stStationEvents[0].aEvents[25].bFault						:= TRUE;
stStationEvents[0].aEvents[25].bEventFlag					:= NOT stMachineStatus.bSystemPowerUp AND dw_T06_EL2904.stTerminalInfo.nTerminal_State <> 8;
stStationEvents[0].aEvents[25].bEventText					:= 'T06_EL2904 card in fault' ;
stStationEvents[0].aEvents[25].sSolution					:= 'Reset System';

stStationEvents[0].aEvents[26].bFault						:= TRUE;
stStationEvents[0].aEvents[26].bEventFlag					:= NOT stMachineStatus.bSystemPowerUp AND dw_T07_EL9410.stTerminalInfo.nTerminal_State <> 8;
stStationEvents[0].aEvents[26].bEventText					:= 'T07_EL9410 card in fault' ;
stStationEvents[0].aEvents[26].sSolution					:= 'Reset System';

stStationEvents[0].aEvents[27].bFault						:= TRUE;
stStationEvents[0].aEvents[27].bEventFlag					:= NOT stMachineStatus.bSystemPowerUp AND dw_T08_EL1809.stTerminalInfo.nTerminal_State <> 8;
stStationEvents[0].aEvents[27].bEventText					:= 'T08_EL1809 card in fault' ;
stStationEvents[0].aEvents[27].sSolution					:= 'Reset System';

stStationEvents[0].aEvents[28].bFault						:= TRUE;
stStationEvents[0].aEvents[28].bEventFlag					:= NOT stMachineStatus.bSystemPowerUp AND dw_T09_EL2809.stTerminalInfo.nTerminal_State <> 8;
stStationEvents[0].aEvents[28].bEventText					:= 'T09_EL2809 card in fault' ;
stStationEvents[0].aEvents[28].sSolution					:= 'Reset System';

stStationEvents[0].aEvents[29].bFault						:= TRUE;
stStationEvents[0].aEvents[29].bEventFlag					:= NOT stMachineStatus.bSystemPowerUp AND dw_T10_EL3058.stTerminalInfo.nTerminal_State <> 8;
stStationEvents[0].aEvents[29].bEventText					:= 'T10_EL3058 card in fault' ;
stStationEvents[0].aEvents[29].sSolution					:= 'Reset System';

stStationEvents[0].aEvents[30].bFault						:= TRUE;
stStationEvents[0].aEvents[30].bEventFlag					:= NOT stMachineStatus.bSystemPowerUp AND dw_T11_EL1918.stTerminalInfo.nTerminal_State <> 8;
stStationEvents[0].aEvents[30].bEventText					:= 'T11_EL1918 card in fault' ;
stStationEvents[0].aEvents[30].sSolution					:= 'Reset System';

stStationEvents[0].aEvents[31].bFault						:= TRUE;
stStationEvents[0].aEvents[31].bEventFlag					:= NOT stMachineStatus.bSystemPowerUp AND dw_T12_EL6633.stTerminalInfo.nTerminal_State <> 8 AND NOT abMachineDefinition[2];
stStationEvents[0].aEvents[31].bEventText					:= 'T12_EL6633 card in fault' ;
stStationEvents[0].aEvents[31].sSolution					:= 'Reset System';

//GENERAL
stStationEvents[0].aEvents[32].bFault						:= TRUE;
stStationEvents[0].aEvents[32].bEventFlag					:= bDoorClosingFlag AND (NOT dw_T05_EL1918.iLeftTouchButtonNO OR NOT dw_T05_EL1918.iRightTouchButtonNO);
stStationEvents[0].aEvents[32].bEventText					:= 'Hands out before door was closed' ;
stStationEvents[0].aEvents[32].sSolution					:= 'Reset System';

stStationEvents[0].aEvents[33].bFault						:= TRUE;
stStationEvents[0].aEvents[33].bEventFlag					:= ((stMachineStatus.eMachineState = E_MachineState.MANUAL_MODE) OR (stMachineStatus.eMachineState = E_MachineState.SYSTEM_AUTO_CYCLE ))
																AND bOutHMI;
stStationEvents[0].aEvents[33].bEventText					:= 'Out HMI while Machine was in Autocycle' ;
stStationEvents[0].aEvents[33].sSolution					:= 'Reset System';


stStationEvents[0].aEvents[34].bFault						:= TRUE;
stStationEvents[0].aEvents[34].bEventTimer(IN := (stMachineStatus.eMachineState = E_MachineState.SYSTEM_AUTO_CYCLE) AND NOT bAutocycleIDLE, PT := stTimers.tAutoCycleTimeOut );
stStationEvents[0].aEvents[34].bEventFlag					:= stStationEvents[0].aEvents[34].bEventTimer.Q;
stStationEvents[0].aEvents[34].bEventText					:= 'Auto Cycle Timeout' ;
stStationEvents[0].aEvents[34].sSolution					:= 'Reset System';

// PUCK LOCKER //Renan Added 06Jul26
stStationEvents[0].aEvents[35].bFault := stMACHINE.bPuckLocker;
stStationEvents[0].aEvents[35].bEventFlag := stMACHINE.bPuckLocker AND GVL_Stations.stPuckLocker.bUnexpectedRemovalFault;
stStationEvents[0].aEvents[35].bEventText := 'Puck removed while locker pin was engaged';
stStationEvents[0].aEvents[35].sSolution := 'Return puck to the locker position and acknowledge the alarm with Administrator access';





//STOP REQUEST

stStationEvents[0].aEvents[40].bCycleStopRequest			:= TRUE;
stStationEvents[0].aEvents[40].bEventFlag					:=  bOutHMI;
stStationEvents[0].aEvents[40].bEventText					:= 'Out HMI or User not logged in' ;
stStationEvents[0].aEvents[40].sSolution					:= '';

stStationEvents[0].aEvents[41].bCycleStopRequest			:= TRUE;
stStationEvents[0].aEvents[41].bEventTimer(IN := bAutocycleIDLE, PT := stTimers.tAutoCycleIDLETimeOut);
stStationEvents[0].aEvents[41].bEventFlag					:= stStationEvents[0].aEvents[41].bEventTimer.Q;
stStationEvents[0].aEvents[41].bEventText					:= 'Autocycle in IDLE Timeout' ;
stStationEvents[0].aEvents[41].sSolution					:= '';

stStationEvents[0].aEvents[42].bCycleStopRequest			:= TRUE;
stStationEvents[0].aEvents[42].bEventFlag					:= NOT dw_T08_EL1809.iStopButton;
stStationEvents[0].aEvents[42].bEventText					:= 'Stop Button Pressed' ;
stStationEvents[0].aEvents[42].sSolution					:= '';

stStationEvents[0].aEvents[43].bCycleStopRequest			:= TRUE;
stStationEvents[0].aEvents[43].bEventFlag					:=  stTwinSAFE.qMainDoorOpenned;
stStationEvents[0].aEvents[43].bEventText					:= 'Door openned ' ;
stStationEvents[0].aEvents[43].sSolution					:= 'Close door and Reset system to intilisation';


stStationEvents[0].aEvents[44].bCycleStopRequest			:= TRUE;
stStationEvents[0].aEvents[44].bEventFlag					:=  (stMachineStatus.eMachineState = E_MachineState.SYSTEM_AUTO_CYCLE) AND NOT bNest1Flag AND NOT bNest2Flag;
stStationEvents[0].aEvents[44].bEventText					:= 'No Nest enabled' ;
stStationEvents[0].aEvents[44].sSolution					:= 'Enable at least one Nest';


//MESSAGES

stStationEvents[0].aEvents[60].bMessage						:= TRUE;
stStationEvents[0].aEvents[60].bEventFlag					:=  bCSVError;
stStationEvents[0].aEvents[60].bEventText					:= 'CSV Not written ' ;
stStationEvents[0].aEvents[60].sSolution					:= '';
END_ACTION

END_PROGRAM

// ---- POUs/C_HMI/C_1_PRG_MainHMI.TcPOU
PROGRAM C_1_PRG_MainHMI
VAR
	
	bResetTest				: BOOL;
	i						: DINT;
	n						: DINT;//TABLE INDEX
	
	srRejectChuteFull			: SR; 

END_VAR

a_ACT_MachineStatusBaner();
b_ACT_Timers();
c_ACT_IO();

bEnableSettings				:= (stMachineStatus.eMachineState = E_MachineState.STOPPED);

stStatisticsWH[0]			:= stStatisticsHMI[0];
stStatisticsWH[1]			:= stStatisticsHMI[1];
stStatisticsWH[2]			:= stStatisticsHMI[4];
stStatisticsWH[3]			:= stStatisticsHMI[5];
stStatisticsWH[4]			:= stStatisticsHMI[6];
stStatisticsWH[5]			:= stStatisticsHMI[7];

stStatisticsLT[0]			:= stStatisticsHMI[0];
stStatisticsLT[1]			:= stStatisticsHMI[1];
stStatisticsLT[2]			:= stStatisticsHMI[2];
stStatisticsLT[3]			:= stStatisticsHMI[3];

bOpenRejectDialog			:= bRejectPartDialog[0] OR bRejectPartDialog[1] OR bRejectPartDialog[2];

bProcessCylinderDownEnable	:= dw_T08_EL1809.iPartPresentNest1 AND dw_T08_EL1809.iPartPresentNest2 AND dw_T05_EL1918.iProcessDoorFB;

srRejectChuteFull(SET1 := stStationEvents[0].aEvents[18].bEventTimer.Q, RESET := bEmptyRejectChuteAcknowledge AND NOT dw_T08_EL1809.iRejectSensor , Q1 => bEmptyRejectChute);

ACTION a_ACT_MachineStatusBaner:
//Machine status banner action
//SYSTEM POWER UP
IF stMachineStatus.bSystemPowerUp THEN	
	stStatusBanner.sMachineStatusText 							:= 'SYSTEM POWER UP';	
	stStatusBanner.nMachineStatusColour 						:= nWHITE;
	stStatusBanner.nMachineStatusTxtCol 						:= nBLACK;
	stStatusBanner.sBannerBckColor 								:= sWHITE;
	stStatusBanner.sBannerTextColor 							:= sBLACK;
END_IF

(* SYSTEM INITIALISING *)
IF stMachineStatus.bInitialising THEN	
	stStatusBanner.sMachineStatusText 							:= 'SYSTEM INITIALIZING';		
	stStatusBanner.nMachineStatusColour 						:= nYELLOW;
	stStatusBanner.nMachineStatusTxtCol 						:= nBLACK;
	stStatusBanner.sBannerBckColor 								:= sYELLOW;
	stStatusBanner.sBannerTextColor 							:= sBLACK;
END_IF

(* SAFETY *)
IF stMachineStatus.bSafety THEN	
	stStatusBanner.sMachineStatusText 							:= 'SYSTEM INITIALIZING';		
	stStatusBanner.nMachineStatusColour 						:= nYELLOW;
	stStatusBanner.nMachineStatusTxtCol 						:= nBLACK;
	stStatusBanner.sBannerBckColor 								:= sYELLOW;
	stStatusBanner.sBannerTextColor 							:= sBLACK;
END_IF


(* SYSTEM READY TO START FLASH ON *)
IF stMachineStatus.bReadyToStart AND stPuls.bFlash1Hz THEN
	stStatusBanner.sMachineStatusText 							:= 'SYSTEM READY TO START';		
	stStatusBanner.nMachineStatusColour 						:= nGREEN;
	stStatusBanner.nMachineStatusTxtCol 						:= nWHITE;
	stStatusBanner.sBannerBckColor 								:= sGREEN;
	stStatusBanner.sBannerTextColor 							:= sWHITE;
ELSIF stMachineStatus.bReadyToStart AND NOT stPuls.bFlash1Hz THEN	
	stStatusBanner.sMachineStatusText 							:= 'SYSTEM READY TO START';		
	stStatusBanner.nMachineStatusColour 						:= nWHITE;
	stStatusBanner.nMachineStatusTxtCol 						:= nGREEN;
	stStatusBanner.sBannerBckColor 								:= sWHITE;
	stStatusBanner.sBannerTextColor 							:= sGREEN;
END_IF

(* SYSTEM AUTO CYCLE *)
IF stMachineStatus.bAutoCycle THEN	
	stStatusBanner.sMachineStatusText 							:= 'SYSTEM AUTO CYCLE';		
	stStatusBanner.nMachineStatusColour 						:= nGREEN;
	stStatusBanner.nMachineStatusTxtCol 						:= nWHITE;
	stStatusBanner.sBannerBckColor 								:= sGREEN;
	stStatusBanner.sBannerTextColor 							:= sWHITE;	
END_IF

(* STOPPING *)
IF stMachineStatus.bStopping AND stPuls.bFlash1Hz THEN	
	stStatusBanner.sMachineStatusText 							:= 'STOPPING';		
	stStatusBanner.nMachineStatusColour 						:= nBLACK;
	stStatusBanner.nMachineStatusTxtCol 						:= nWHITE;
	stStatusBanner.sBannerBckColor 								:= sBLACK;
	stStatusBanner.sBannerTextColor 							:= sWHITE;	
ELSIF stMachineStatus.bStopping AND NOT stPuls.bFlash1Hz THEN	
	stStatusBanner.sMachineStatusText 							:= 'STOPPING';		
	stStatusBanner.nMachineStatusColour 						:= nWHITE;
	stStatusBanner.nMachineStatusTxtCol 						:= nBLACK;
	stStatusBanner.sBannerBckColor 								:= sWHITE;
	stStatusBanner.sBannerTextColor 							:= sBLACK;	
END_IF

(*STOPPED *)
IF stMachineStatus.bStopped THEN	
	stStatusBanner.sMachineStatusText 							:= 'CYCLE STOPPED';		
	stStatusBanner.nMachineStatusColour 						:= nBLACK;
	stStatusBanner.nMachineStatusTxtCol 						:= nWHITE;
	stStatusBanner.sBannerBckColor 								:= sBLACK;
	stStatusBanner.sBannerTextColor 							:= sWHITE;	
END_IF

(* FAULT FLASH ON *)
IF stMachineStatus.bFault AND stPuls.bFlash1Hz THEN	
	stStatusBanner.sMachineStatusText 							:= 'FAULT';		
	stStatusBanner.nMachineStatusColour 						:= nRED;
	stStatusBanner.nMachineStatusTxtCol 						:= nWHITE;
	stStatusBanner.sBannerBckColor 								:= sRED;
	stStatusBanner.sBannerTextColor 							:= sWHITE;	
ELSIF stMachineStatus.bFault AND NOT stPuls.bFlash1Hz THEN	
	stStatusBanner.sMachineStatusText 							:= 'FAULT';		
	stStatusBanner.nMachineStatusColour 						:= nWHITE;
	stStatusBanner.nMachineStatusTxtCol 						:= nBLACK;
	stStatusBanner.sBannerBckColor 								:= sWHITE;
	stStatusBanner.sBannerTextColor 							:= sBLACK;	
END_IF

(* MANUAL MODE *)
IF stMachineStatus.bManualMode THEN	
	stStatusBanner.sMachineStatusText 							:= 'MANUAL MODE';		
	stStatusBanner.nMachineStatusColour 						:= nBLUE;
	stStatusBanner.nMachineStatusTxtCol 						:= nWHITE;
	stStatusBanner.sBannerBckColor 								:= sBLUE;
	stStatusBanner.sBannerTextColor 							:= sWHITE;	
END_IF
END_ACTION

ACTION b_ACT_Timers:

stTimers.tAutoCycleTimeOut		:= DINT_TO_TIME(stTimers.nAutoCycleTimeOut * 1000) ;
stTimers.tDoorOpenedSignal		:= DINT_TO_TIME(stTimers.nDoorOpenedSignal * 1000) ;
stTimers.tStation1TimeOut		:= DINT_TO_TIME(stTimers.nStation1TimeOut * 1000) ;
stTimers.tStation2TimeOut		:= DINT_TO_TIME(stTimers.nStation2TimeOut * 1000) ;
stTimers.tStation3TimeOut		:= DINT_TO_TIME(stTimers.nStation3TimeOut * 1000) ;
stTimers.tTwoHandsSignal		:= DINT_TO_TIME(stTimers.nTwoHandsSignal * 1000) ;
stTimers.tHeightTest			:= DINT_TO_TIME(stTimers.nHeightTest * 1000) ;
stTimers.tAutoCycleIDLETimeOut			:= DINT_TO_TIME(stTimers.nAutoCycleIDLETimeOut * 1000) ;
END_ACTION

ACTION c_ACT_IO:
dw_T09_EL2809.qPanelLightLED				:= bLightsOnOff;
END_ACTION

END_PROGRAM

// ---- POUs/Utilities/PRG_Puls.TcPOU
PROGRAM PRG_Puls
VAR
	    //=== Master Pulses ===//
	fbScalingFlash  :FB_Pulse;
	fbScalingFlash4 :FB_Pulse;
	fbScalingFlash5 :FB_Pulse;
	fbFlash100Hz    :FB_Pulse;
	fbFlash10Hz		:FB_Pulse;
	fbFlash10HzB    :FB_Pulse;
	fbFlash4Hz		:FB_Pulse;
	fbFlash2Hz		:FB_Pulse;
	fbFlash1Hz		:FB_Pulse;
    fbFlash5Sec     :FB_Pulse;			

END_VAR

    //=== Master Pulses ===//
(**************************************************************************************************)
fbScalingFlash(
	bEnable	:=	TRUE,
	tPulseOn	:=	T#2MS,
	tPulseOff	:=	T#2MS,
	bFlash		=>	stPuls.bFlashScale
);

fbScalingFlash4(
     bEnable	:=	TRUE,
	tPulseOn	:=	T#4MS,
	tPulseOff	:=	T#4MS,
	bFlash		=>	stPuls.bFlashScale4
);
fbScalingFlash5(
     bEnable	:=	TRUE,
	tPulseOn	:=	T#5MS,
	tPulseOff	:=	T#5MS,
	bFlash		=>	stPuls.bFlashScale5
);



fbFlash100Hz(
	bEnable	:=	TRUE,
	tPulseOn	:=	T#10MS,
	tPulseOff	:=	T#10MS,
	bFlash		=>	stPuls.bFlash100Hz
);


fbFlash10HzB ( 
    bEnable	    :=	TRUE,
	tPulseOn	:=	T#20MS,//  T#50MS,
	tPulseOff	:=	T#20MS,//  T#50MS,
	bFlash		=>	stPuls.bFlash10BHz
);


fbFlash10Hz(
	bEnable	:=	TRUE,
	tPulseOn	:=	T#100MS,
	tPulseOff	:=	T#100MS,
	bFlash		=>	stPuls.bFlash10Hz
);


fbFlash4Hz(
	bEnable	:=	TRUE,
	tPulseOn	:=	T#250MS,
	tPulseOff	:=	T#250MS,
	bFlash		=>	stPuls.bFlash4Hz
);

fbFlash2Hz(
	bEnable	:=	TRUE,
	tPulseOn	:=	T#500MS,
	tPulseOff	:=	T#500MS,
	bFlash		=>	stPuls.bFlash2Hz
);

fbFlash1Hz(
	bEnable	:=	TRUE,
	tPulseOn	:=	T#1000MS,
	tPulseOff	:=	T#1000MS,
	bFlash		=>	stPuls.bFlash1Hz
);

fbFlash5Sec(
	bEnable	:=	TRUE,
	tPulseOn	:=	T#5S,
	tPulseOff	:=	T#5S,
	bFlash		=>	stPuls.bFlash5sec
);

END_PROGRAM

// ---- POUs/Utilities/FB_Pulse.TcPOU
FUNCTION_BLOCK FB_Pulse
VAR_INPUT
	bEnable		    :	BOOL;
	tPulseOn		:	TIME;
	tPulseOff		:	TIME;
END_VAR
VAR_OUTPUT
	bFlash			:	BOOL;
END_VAR
VAR
	tonFlashOn		:	TON;
	tonFlashOff	    :	TON;
END_VAR

IF 		(bEnable 	AND NOT 	tonFlashOff.Q)		THEN
	tonFlashOn.IN			:=	TRUE;
ELSE
	tonFlashOn.IN			:=	FALSE;
END_IF

tonFlashOn(
	IN:= ,
	PT:= tPulseOn,
	Q=> ,
	ET=>
);
tonFlashOff(
	IN:= tonFlashOn.Q,
	PT:= tPulseOff,
	Q=> ,
	ET=>
);

bFlash	:=	tonFlashOn.Q;

END_FUNCTION_BLOCK

// ---- POUs/B_STATIONS/B_2_HEIGHT_TEST/B_2_1_PRG_Master_Height_Test.TcPOU
PROGRAM B_2_1_PRG_Master_Height_Test

VAR

	rGoodStatistics						: ARRAY[0..1] OF  R_TRIG;
	rBadStatistics						: ARRAY[0..1] OF  R_TRIG;
	rEfficency							: STRING(510);
	
	anMinimumDistance					: ARRAY[1..3] OF REAL;
	anMaximumDistance					: ARRAY[1..3] OF REAL;

/////////////////////////////////////////////////////////////////////////////////////I O/////////////////////////////////////////////////////////////////////////////////////	
	
	abPass1								: ARRAY [1..3] OF BOOL;
	abFail1								: ARRAY [1..3] OF BOOL;
	abPass2								: ARRAY [1..3] OF BOOL;
	abFail2								: ARRAY [1..3] OF BOOL;
	tonTakeMeasure						: TON;
	abMeaurement						: ARRAY [0..1] OF BOOL;
	bMeasurementDone					: BOOL;

	abProbeError1						: ARRAY[1..4] OF BOOL;
	abProbeError2						: ARRAY[1..4] OF BOOL;
	bGeneralProbeError					: BOOL;
	bGeneralError						: BOOL;
	anRawMesurement1					: ARRAY[1..4] OF REAL;
	anRawMesurement2					: ARRAY[1..4] OF REAL;
	anRealDistance1						: ARRAY[1..3] OF REAL;
	anRealDistance2						: ARRAY[1..3] OF REAL;
	(*Renan - Added on 30Jun2026 *)
	anCorrectedMeasurement1 			: ARRAY [1..4] OF REAL;
    anCorrectedMeasurement2 			: ARRAY [1..4] OF REAL;
	(*/Renan - Added on 30Jun2026 *)

	i									: DINT;
	j									: DINT; //Index for settings
	
	
	

	
END_VAR

d_ACT_Set_Events_Station_2();
a_ACT_Ctrl_Station_2();
b_ACT_IO();
c_ACT_Statistics_Station_2();
e_ACT_Measurement();
f_ACT_ManualMode();
g_ACT_Settings();

ACTION a_ACT_Ctrl_Station_2:
/////////////////////////////////////////////////////////////////////////////////////UTILITIES/////////////////////////////////////////////////////////////////////////////////////
IF bGeneralProbeError OR bGeneralError OR stHeightTests.CMD.bAbort THEN
	
	stHeightTests.State			:= E_HeightTest_State.RESET;

ELSIF stHeightTests.CMD.bManualMode THEN
	
	stHeightTests.State			:= E_HeightTest_State.MANUAL_MODE;
	
END_IF



/////////////////////////////////////////////////////////////////////////////////////CONDITIONS/////////////////////////////////////////////////////////////////////////////////////

CASE stHeightTests.State OF
	
	E_HeightTest_State.ABORTED:

								IF 	stHeightTests.CMD.bEnable THEN
									
									stHeightTests.State			:= E_HeightTest_State.READY;
								
								END_IF
								
								

	E_HeightTest_State.READY:
	
								IF stHeightTests.CMD.bExecute THEN
									
									stHeightTests.State			:= E_HeightTest_State.MEASURE;
								
								END_IF
		
	E_HeightTest_State.MEASURE:				
									
								IF stHeightTests.CMD.HeightTest_CMD.Measurement1 AND stHeightTests.CMD.HeightTest_CMD.Measurement2 THEN
										
									abMeaurement[0]			:= TRUE;
									abMeaurement[1]			:= TRUE;
									
								ELSIF stHeightTests.CMD.HeightTest_CMD.Measurement1 AND NOT stHeightTests.CMD.HeightTest_CMD.Measurement2 THEN
									
									abMeaurement[0]			:= TRUE;
									
								ELSIF NOT stHeightTests.CMD.HeightTest_CMD.Measurement1 AND stHeightTests.CMD.HeightTest_CMD.Measurement2 THEN
									
									abMeaurement[1]			:= TRUE;
									
								END_IF
									
								stHeightTests.State			:= E_HeightTest_State.WAIT_MEASUREMENT;
								
	E_HeightTest_State.WAIT_MEASUREMENT:						
								
								e_ACT_Measurement();
								
								IF stHeightTests.CMD.HeightTest_CMD.Measurement1 THEN
									
									stCycleDataNest1.HeightTest_anRawMeasurement				:= anRawMesurement1;
									stCycleDataNest1.HeightTest_anDistancesResult 				:= anRealDistance1;
									stCycleDataNest1.HeightTest_bDistancesResult				:= abPass1;
									
								END_IF
								IF stHeightTests.CMD.HeightTest_CMD.Measurement2 THEN
									
									stCycleDataNest2.HeightTest_anRawMeasurement				:= anRawMesurement2;																
									stCycleDataNest2.HeightTest_anDistancesResult 				:= anRealDistance2;																
									stCycleDataNest2.HeightTest_bDistancesResult				:= abPass2;
									
								END_IF
								
								
								IF bMeasurementDone THEN
			
									stHeightTests.State		:= E_HeightTest_State.DONE;
								
								END_IF
										
	E_HeightTest_State.DONE:
								IF  stHeightTests.CMD.bAcknowledge THEN
									
									stHeightTests.State									:= E_HeightTest_State.RESULTS;
									stHeightTests.CMD.bAcknowledge 						:= FALSE;
									
								END_IF	
								
	E_HeightTest_State.RESULTS:
							
								IF abMeaurement[0] THEN
									IF abPass1[1] AND abPass1[2] AND abPass1[3] THEN
									
										stCycleDataNest1.HeightTest_Pass				:= TRUE;
									
									ELSE stCycleDataNest1.HeightTest_Fail 				:= TRUE;
								
									END_IF
								END_IF
								
								IF abMeaurement[1] THEN
									IF abPass2[1] AND abPass2[2] AND abPass2[3] THEN
									
										stCycleDataNest2.HeightTest_Pass				:= TRUE;
									
									ELSE stCycleDataNest2.HeightTest_Fail  			:= TRUE;
								
									END_IF
								END_IF	
								
								stHeightTests.State										:= E_HeightTest_State.RESET;
								
	E_HeightTest_State.RESET:
	
								abMeaurement[0]											:= FALSE;
								abMeaurement[1]											:= FALSE;
								bMeasurementDone										:= FALSE;

								FOR i := 1 TO 3 DO
									
									abPass1[i]											:= FALSE;
									abFail1[i]											:= FALSE;
									abPass2[i]											:= FALSE;
									abFail2[i]											:= FALSE;
								
								END_FOR
								
								IF bGeneralProbeError OR bGeneralError THEN
									
									stHeightTests.State									:= E_HeightTest_State.ERROR;
								
								ELSIF stHeightTests.CMD.bAbort THEN
									
									stHeightTests.State									:= E_HeightTest_State.ABORTED;
								
								ELSE stHeightTests.State								:= E_HeightTest_State.READY;
									
								END_IF
								
								
	
	E_HeightTest_State.ERROR:
	
								IF NOT bGeneralProbeError OR bGeneralError THEN
									
									stHeightTests.State									:= E_HeightTest_State.RESET;
									
								END_IF
							
	E_HeightTest_State.MANUAL_MODE:
	
								f_ACT_ManualMode();
								
								IF NOT stHeightTests.CMD.bManualMode THEN
									
									stHeightTests.State									:= E_HeightTest_State.ABORTED;
									
								END_IF
								
	
								

ELSE stHeightTests.State := E_HeightTest_State.READY;
	
END_CASE
/////////////////////////////////////////////////////////////////////////////////////STATUS/////////////////////////////////////////////////////////////////////////////////////

stHeightTests.Status.bBusy	:= 	stHeightTests.State	= E_HeightTest_State.WAIT_MEASUREMENT;	

stHeightTests.Status.bDone	:= 	stHeightTests.State	= E_HeightTest_State.DONE;

stHeightTests.Status.bError	:= 	stHeightTests.State	= E_HeightTest_State.ERROR;	

stHeightTests.Status.bReady	:=	stHeightTests.State	= E_HeightTest_State.READY;

stHeightTests.Status.bStopped := NOT stHeightTests.Status.bBusy;
END_ACTION

ACTION b_ACT_IO:

	abProbeError1					:= Probes.stProbesSet[1].abProbeError;
	abProbeError2					:= Probes.stProbesSet[2].abProbeError;
	bGeneralError					:= Probes.bGeneralError;
	anRawMesurement1				:= Probes.stProbesSet[1].anScaledRawMeasurement;
	anRawMesurement2				:= Probes.stProbesSet[2].anScaledRawMeasurement;
	


	bGeneralProbeError				:= 	abProbeError1[1] OR abProbeError1[2] OR abProbeError1[3] OR abProbeError1[4] OR
										abProbeError2[1] OR abProbeError2[2] OR abProbeError2[3] OR abProbeError2[4];
										
	stCycleDataNest1.HeightTest_anSetPoint := stProbesSettings.anExpectedDistances;
	stCycleDataNest2.HeightTest_anSetPoint := stProbesSettings.anExpectedDistances;
END_ACTION

ACTION c_ACT_Statistics_Station_2:
stStatisticsHMI[4].sName			:= 'Height Test 1';
stStatisticsHMI[5].sName			:= 'Height Test 2';


rGoodStatistics[0]( CLK := stCycleDataNest1.HeightTest_Pass);
rGoodStatistics[1]( CLK := stCycleDataNest2.HeightTest_Pass);
rBadStatistics[0]	( CLK := stCycleDataNest1.HeightTest_Fail);
rBadStatistics[1]	( CLK := stCycleDataNest2.HeightTest_Fail);

//statistics 1
IF 	rGoodStatistics[0].Q THEN
	
	stStatisticsHMI[4].nGood		:= stStatisticsHMI[4].nGood + 1;
	
END_IF
								
IF 	rBadStatistics[0].Q THEN
	
	stStatisticsHMI[4].nBad			:= stStatisticsHMI[4].nBad + 1;
	
END_IF

IF stStatisticsHMI[4].bResetGood THEN
	stStatisticsHMI[4].nGood		:= 0;
END_IF

IF stStatisticsHMI[4].bResetBad THEN
	stStatisticsHMI[4].nBad			:= 0;
END_IF

IF (( stStatisticsHMI[4].nGood + stStatisticsHMI[4].nBad) <> 0) THEN
	
	rEfficency							:= LREAL_TO_FMTSTR(in := (DINT_TO_REAL(stStatisticsHMI[4].nGood) /( DINT_TO_REAL(stStatisticsHMI[4].nGood) + DINT_TO_REAL(stStatisticsHMI[4].nBad))) * 100.0,iPrecision := 2, bRound := TRUE);
	stStatisticsHMI[4].nEfficency		:= CONCAT(STR1 := '%', STR2 := (rEfficency));

ELSE stStatisticsHMI[4].nEfficency		:= CONCAT(STR1 := '%', STR2 := (DINT_TO_STRING(0)));
	
END_IF
//statistics 2
IF 	rGoodStatistics[1].Q THEN
	
	stStatisticsHMI[5].nGood		:= stStatisticsHMI[5].nGood + 1;
	
END_IF
								
IF 	rBadStatistics[1].Q THEN
	
	stStatisticsHMI[5].nBad			:= stStatisticsHMI[5].nBad + 1;
	
END_IF

IF stStatisticsHMI[5].bResetGood THEN
	stStatisticsHMI[5].nGood		:= 0;
END_IF

IF stStatisticsHMI[5].bResetBad THEN
	stStatisticsHMI[5].nBad			:= 0;
END_IF

IF (( stStatisticsHMI[5].nGood + stStatisticsHMI[5].nBad) <> 0) THEN
	
	rEfficency							:= LREAL_TO_FMTSTR(in := (DINT_TO_REAL(stStatisticsHMI[5].nGood) /( DINT_TO_REAL(stStatisticsHMI[5].nGood) + DINT_TO_REAL(stStatisticsHMI[5].nBad))) * 100.0,iPrecision := 2, bRound := TRUE);
	stStatisticsHMI[5].nEfficency		:= CONCAT(STR1 := '%', STR2 := (rEfficency));

ELSE stStatisticsHMI[5].nEfficency		:= CONCAT(STR1 := '%', STR2 := (DINT_TO_STRING(0)));
	
END_IF
END_ACTION

ACTION d_ACT_Set_Events_Station_2:
//FAULTS

stStationEvents[2].aEvents[0].bFault						:= TRUE;
stStationEvents[2].aEvents[0].bEventFlag					:= bGeneralError;
stStationEvents[2].aEvents[0].bEventText					:= 'Probes general error';
stStationEvents[2].aEvents[0].sSolution						:= 'Check probes amplifier and ethercat unit';

stStationEvents[2].aEvents[1].bFault						:= TRUE;
stStationEvents[2].aEvents[1].bEventFlag					:= abProbeError1[1];
stStationEvents[2].aEvents[1].bEventText					:= 'Probes 1 error';
stStationEvents[2].aEvents[1].sSolution						:= 'Check probe 1';

stStationEvents[2].aEvents[2].bFault						:= TRUE;
stStationEvents[2].aEvents[2].bEventFlag					:= abProbeError1[2];
stStationEvents[2].aEvents[2].bEventText					:= 'Probes 2 error';
stStationEvents[2].aEvents[2].sSolution						:= 'Check probe 2';

stStationEvents[2].aEvents[3].bFault						:= TRUE;
stStationEvents[2].aEvents[3].bEventFlag					:= abProbeError1[3];
stStationEvents[2].aEvents[3].bEventText					:= 'Probes 3 error';
stStationEvents[2].aEvents[3].sSolution						:= 'Check probe 3';

stStationEvents[2].aEvents[4].bFault						:= TRUE;
stStationEvents[2].aEvents[4].bEventFlag					:= abProbeError1[4];
stStationEvents[2].aEvents[4].bEventText					:= 'Probes 4 error';
stStationEvents[2].aEvents[4].sSolution						:= 'Check probe 4';

stStationEvents[2].aEvents[5].bFault						:= TRUE;
stStationEvents[2].aEvents[5].bEventFlag					:= abProbeError2[1];
stStationEvents[2].aEvents[5].bEventText					:= 'Probes 5 error';
stStationEvents[2].aEvents[5].sSolution						:= 'Check probe 5';

stStationEvents[2].aEvents[6].bFault						:= TRUE;
stStationEvents[2].aEvents[6].bEventFlag					:= abProbeError2[2];
stStationEvents[2].aEvents[6].bEventText					:= 'Probes 6 error';
stStationEvents[2].aEvents[6].sSolution						:= 'Check probe 6';

stStationEvents[2].aEvents[7].bFault						:= TRUE;
stStationEvents[2].aEvents[7].bEventFlag					:= abProbeError2[3];
stStationEvents[2].aEvents[7].bEventText					:= 'Probes 7 error';
stStationEvents[2].aEvents[7].sSolution						:= 'Check probe 7';

stStationEvents[2].aEvents[8].bFault						:= TRUE;
stStationEvents[2].aEvents[8].bEventFlag					:= abProbeError2[4];
stStationEvents[2].aEvents[8].bEventText					:= 'Probes 8 error';
stStationEvents[2].aEvents[8].sSolution						:= 'Check probe 8';

stStationEvents[2].aEvents[9].bFault						:= TRUE;
stStationEvents[2].aEvents[9].bEventTimer(IN := stHeightTests.Status.bBusy, PT := stTimers.tStation2TimeOut);
stStationEvents[2].aEvents[9].bEventFlag					:= stStationEvents[2].aEvents[9].bEventTimer.Q;
stStationEvents[2].aEvents[9].bEventText					:= 'Height test cycle Timeout';
stStationEvents[2].aEvents[9].sSolution						:= 'Reset System';
END_ACTION

ACTION e_ACT_Measurement:

tonTakeMeasure(IN:= stHeightTests.State = E_HeightTest_State.WAIT_MEASUREMENT, PT := stTimers.tHeightTest);

IF tonTakeMeasure.Q THEN
	
	IF abMeaurement[0] THEN
	
		FOR i := 1 TO 3 DO
		
			IF (anRealDistance1[i] > anMinimumDistance[i]) AND (anRealDistance1[i] < anMaximumDistance[i]) THEN
		
				abPass1[i]						:= TRUE;
			
			ELSE abFail1[i]						:= TRUE;	
				
			END_IF
		
		END_FOR

	END_IF
	
	IF abMeaurement[1] THEN
	
		FOR i := 1 TO 3 DO
		
			IF (anRealDistance2[i] > anMinimumDistance[i]) AND (anRealDistance2[i] < anMaximumDistance[i]) THEN
		
				abPass2[i]						:= TRUE;
			
			ELSE abFail2[i]						:= TRUE;	
				
			END_IF
		
		END_FOR

	END_IF

	bMeasurementDone							:= TRUE;
	i											:= 0;
END_IF
END_ACTION

ACTION f_ACT_ManualMode:
IF stPuls.bFlash100Hz THEN
	
	FOR i := 1 TO 3 DO
		
		IF (anRealDistance1[i] > anMinimumDistance[i]) AND (anRealDistance1[i] < anMaximumDistance[i]) THEN
		
			stAnimations.abDistanceBoxesGreen[i]	:= TRUE;
			
		ELSE stAnimations.abDistanceBoxesGreen[i]	:= FALSE;	
				
		END_IF
		
	END_FOR
	i												:= 0;
	FOR i := 1 TO 3 DO
		
		IF (anRealDistance2[i] > anMinimumDistance[i]) AND (anRealDistance2[i] < anMaximumDistance[i]) THEN
		
			stAnimations.abDistanceBoxesGreen[3+i]	:= TRUE;
			
		ELSE stAnimations.abDistanceBoxesGreen[3+i]	:= FALSE;	
				
		END_IF
		
	END_FOR
	
	i												:= 0;
END_IF
END_ACTION

ACTION g_ACT_Settings:
//settings tolerances

anMinimumDistance[1]					:= stProbesSettings.anExpectedDistances[1] - stProbesSettings.anTolerances[1];//settings from HMI
anMaximumDistance[1]					:= stProbesSettings.anExpectedDistances[1] + stProbesSettings.anTolerances[1];//settings from HMI
anMinimumDistance[2]					:= stProbesSettings.anExpectedDistances[2] - stProbesSettings.anTolerances[2];//settings from HMI
anMaximumDistance[2]					:= stProbesSettings.anExpectedDistances[2] + stProbesSettings.anTolerances[2];//settings from HMI
anMinimumDistance[3]					:= stProbesSettings.anExpectedDistances[3] - stProbesSettings.anTolerances[3];//settings from HMI
anMaximumDistance[3]					:= stProbesSettings.anExpectedDistances[3] + stProbesSettings.anTolerances[3];//settings from HMI





//setting the bit according to the probe from bit 1 to bit 8
IF abPresetProbe[1] THEN
	
	Probes.abPresetProbe						:= 2;

ELSIF abPresetProbe[2] THEN
	
	Probes.abPresetProbe						:= 4;
	
ELSIF abPresetProbe[3] THEN
	
	Probes.abPresetProbe						:= 8;
	
ELSIF abPresetProbe[4] THEN
	
	Probes.abPresetProbe						:= 16;
	
ELSIF abPresetProbe[5] THEN
	
	Probes.abPresetProbe						:= 32;
	
ELSIF abPresetProbe[6] THEN
	
	Probes.abPresetProbe						:= 64;
	
ELSIF abPresetProbe[7] THEN
	
	Probes.abPresetProbe						:= 128;
	
ELSIF abPresetProbe[8] THEN
	
	Probes.abPresetProbe						:= 256;

END_IF

Probes.stProbesSet[1].anScaledRawMeasurement[1]					:= DINT_TO_REAL(Probes.stProbesSet[1].anRawMeasurement[1])/10000;
Probes.stProbesSet[1].anScaledRawMeasurement[2]					:= DINT_TO_REAL(Probes.stProbesSet[1].anRawMeasurement[2])/10000;
Probes.stProbesSet[1].anScaledRawMeasurement[3]					:= DINT_TO_REAL(Probes.stProbesSet[1].anRawMeasurement[3])/10000;
Probes.stProbesSet[1].anScaledRawMeasurement[4]					:= DINT_TO_REAL(Probes.stProbesSet[1].anRawMeasurement[4])/10000;

Probes.stProbesSet[2].anScaledRawMeasurement[1]					:= DINT_TO_REAL(Probes.stProbesSet[2].anRawMeasurement[1])/10000;
Probes.stProbesSet[2].anScaledRawMeasurement[2]					:= DINT_TO_REAL(Probes.stProbesSet[2].anRawMeasurement[2])/10000;
Probes.stProbesSet[2].anScaledRawMeasurement[3]					:= DINT_TO_REAL(Probes.stProbesSet[2].anRawMeasurement[3])/10000;
Probes.stProbesSet[2].anScaledRawMeasurement[4]					:= DINT_TO_REAL(Probes.stProbesSet[2].anRawMeasurement[4])/10000;

IF Probes.stProbesSet[1].anScaledRawMeasurement[1] > 2 AND Probes.stProbesSet[1].anScaledRawMeasurement[1] < 12 AND 
	Probes.stProbesSet[1].anScaledRawMeasurement[2] > 2 AND Probes.stProbesSet[1].anScaledRawMeasurement[2] < 12 AND 
	Probes.stProbesSet[1].anScaledRawMeasurement[3] > 2 AND Probes.stProbesSet[1].anScaledRawMeasurement[3] < 12 AND 
	Probes.stProbesSet[1].anScaledRawMeasurement[4] > 2 AND Probes.stProbesSet[1].anScaledRawMeasurement[4] < 12 THEN 
	
	bEnableSetCablibrationBlock1								:= TRUE;
	
ELSE bEnableSetCablibrationBlock1								:= FALSE;
	
END_IF

IF Probes.stProbesSet[2].anScaledRawMeasurement[1] > 2 AND Probes.stProbesSet[2].anScaledRawMeasurement[1] < 12 AND 
	Probes.stProbesSet[2].anScaledRawMeasurement[2] > 2 AND Probes.stProbesSet[2].anScaledRawMeasurement[2] < 12 AND 
	Probes.stProbesSet[2].anScaledRawMeasurement[3] > 2 AND Probes.stProbesSet[2].anScaledRawMeasurement[3] < 12 AND 
	Probes.stProbesSet[2].anScaledRawMeasurement[4] > 2 AND Probes.stProbesSet[2].anScaledRawMeasurement[4] < 12 THEN 
	
	bEnableSetCablibrationBlock2								:= TRUE;
	
ELSE bEnableSetCablibrationBlock2								:= FALSE;
	
END_IF

//calibration block
IF bSetCalibrationBlock1 THEN
	
	stProbesSettings.anHeightSetByCalibration1[1]				:= Probes.stProbesSet[1].anScaledRawMeasurement[1];
	stProbesSettings.anHeightSetByCalibration1[2]				:= Probes.stProbesSet[1].anScaledRawMeasurement[2];
	stProbesSettings.anHeightSetByCalibration1[3]				:= Probes.stProbesSet[1].anScaledRawMeasurement[3];
	stProbesSettings.anHeightSetByCalibration1[4]				:= Probes.stProbesSet[1].anScaledRawMeasurement[4];
	
	stProbesSettings.nDistanceOffset1[1]						:= stProbesSettings.anDistanceCalibrationBlock[1] - (Probes.stProbesSet[1].anScaledRawMeasurement[2] - Probes.stProbesSet[1].anScaledRawMeasurement[1]);
	stProbesSettings.nDistanceOffset1[2]						:= stProbesSettings.anDistanceCalibrationBlock[2] - (Probes.stProbesSet[1].anScaledRawMeasurement[3] - Probes.stProbesSet[1].anScaledRawMeasurement[1]);
	stProbesSettings.nDistanceOffset1[3]						:= stProbesSettings.anDistanceCalibrationBlock[3] - (Probes.stProbesSet[1].anScaledRawMeasurement[4] - Probes.stProbesSet[1].anScaledRawMeasurement[1]);
	
END_IF



IF bSetCalibrationBlock2 THEN
	
	stProbesSettings.anHeightSetByCalibration2[1]				:= Probes.stProbesSet[2].anScaledRawMeasurement[1];
	stProbesSettings.anHeightSetByCalibration2[2]				:= Probes.stProbesSet[2].anScaledRawMeasurement[2];
	stProbesSettings.anHeightSetByCalibration2[3]				:= Probes.stProbesSet[2].anScaledRawMeasurement[3];
	stProbesSettings.anHeightSetByCalibration2[4]				:= Probes.stProbesSet[2].anScaledRawMeasurement[4];
	
	stProbesSettings.nDistanceOffset2[1]						:= stProbesSettings.anDistanceCalibrationBlock[1] - (Probes.stProbesSet[2].anScaledRawMeasurement[2] - Probes.stProbesSet[2].anScaledRawMeasurement[1]);
	stProbesSettings.nDistanceOffset2[2]						:= stProbesSettings.anDistanceCalibrationBlock[2] - (Probes.stProbesSet[2].anScaledRawMeasurement[3] - Probes.stProbesSet[2].anScaledRawMeasurement[1]);
	stProbesSettings.nDistanceOffset2[3]						:= stProbesSettings.anDistanceCalibrationBlock[3] - (Probes.stProbesSet[2].anScaledRawMeasurement[4] - Probes.stProbesSet[2].anScaledRawMeasurement[1]);

END_IF

(* Renan Added 30Jun26 - Nest offset by probe *)
IF bSetProbeOffsetNest1 THEN
	FOR i := 1 TO 4 DO
		stProbesSettings.anNestOffsetByProbe1[i] := anNestOffsetByProbe1[i];
		stProbesSettings.anNestOffsetByProbe2[i] := anNestOffsetByProbe2[i];
	END_FOR
	bSetProbeOffsetNest1 := FALSE;
END_IF

FOR i := 1 TO 4 DO
    anCorrectedMeasurement1[i] := Probes.stProbesSet[1].anScaledRawMeasurement[i] + stProbesSettings.anNestOffsetByProbe1[i];
    anCorrectedMeasurement2[i] := Probes.stProbesSet[2].anScaledRawMeasurement[i] + stProbesSettings.anNestOffsetByProbe2[i];
END_FOR

(* Renan Changed 30Jun26 - Nest offset by probe *)

anRealDistance1[1] 	:= (anCorrectedMeasurement1[2] - anCorrectedMeasurement1[1]) + stProbesSettings.nDistanceOffset1[1]; //(Probes.stProbesSet[1].anScaledRawMeasurement[2] - Probes.stProbesSet[1].anScaledRawMeasurement[1]) + stProbesSettings.nDistanceOffset1[1];
anRealDistance1[2] 	:= (anCorrectedMeasurement1[3] - anCorrectedMeasurement1[1]) + stProbesSettings.nDistanceOffset1[2]; //(Probes.stProbesSet[1].anScaledRawMeasurement[3] - Probes.stProbesSet[1].anScaledRawMeasurement[1]) + stProbesSettings.nDistanceOffset1[2];
anRealDistance1[3] 	:= (anCorrectedMeasurement1[4] - anCorrectedMeasurement1[1]) + stProbesSettings.nDistanceOffset1[3]; //(Probes.stProbesSet[1].anScaledRawMeasurement[4] - Probes.stProbesSet[1].anScaledRawMeasurement[1]) + stProbesSettings.nDistanceOffset1[3];

anRealDistance2[1] 	:= (anCorrectedMeasurement2[2] - anCorrectedMeasurement2[1]) + stProbesSettings.nDistanceOffset2[1]; //(Probes.stProbesSet[2].anScaledRawMeasurement[2] - Probes.stProbesSet[2].anScaledRawMeasurement[1]) + stProbesSettings.nDistanceOffset2[1];
anRealDistance2[2] 	:= (anCorrectedMeasurement2[3] - anCorrectedMeasurement2[1]) + stProbesSettings.nDistanceOffset2[2]; //(Probes.stProbesSet[2].anScaledRawMeasurement[3] - Probes.stProbesSet[2].anScaledRawMeasurement[1]) + stProbesSettings.nDistanceOffset2[2];
anRealDistance2[3] 	:= (anCorrectedMeasurement2[4] - anCorrectedMeasurement2[1]) + stProbesSettings.nDistanceOffset2[3]; //(Probes.stProbesSet[2].anScaledRawMeasurement[4] - Probes.stProbesSet[2].anScaledRawMeasurement[1]) + stProbesSettings.nDistanceOffset2[3];
END_ACTION

END_PROGRAM

// ---- POUs/B_STATIONS/B_1_LEAK_TEST/B_1_1_PRG_Master_Leak_Test.TcPOU
PROGRAM B_1_1_PRG_Master_Leak_Test

VAR

	tonStationStopped					: TON;
	tonExecute							: TON;
	rGoodStatistics						: ARRAY [0..1] OF R_TRIG;
	rBadStatistics						: ARRAY [0..1] OF R_TRIG;
	rEfficency							: ARRAY [0..1] OF STRING(510);
	
	tonWaitResults						: TON;
/////////////////////////////////////////////////////////////////////////////////////I O/////////////////////////////////////////////////////////////////////////////////////	

	bStopped							: ARRAY [0..1] OF BOOL;
	bError								: ARRAY [0..1] OF BOOL;
	bReady								: ARRAY [0..1] OF BOOL;
	bDone								: ARRAY [0..1] OF BOOL;
	bReset								: ARRAY [0..1] OF BOOL;
	bStart								: ARRAY [0..1] OF BOOL;
	bStop								: ARRAY [0..1] OF BOOL;	
	bBusy								: ARRAY [0..1] OF BOOL;	
	fLeakTestDone						: ARRAY [0..1] OF F_TRIG;	
	bLeakTestDone						: ARRAY [0..1] OF BOOL;	
	rPass								: ARRAY [0..1] OF R_TRIG;	
	bPass								: ARRAY [0..1] OF BOOL;	
	rFail								: ARRAY [0..1] OF R_TRIG;	
	bFail								: ARRAY [0..1] OF BOOL;
	rReset								: ARRAY [0..1] OF R_TRIG;

	
END_VAR

a_ACT_Ctrl_Station_1();
b_ACT_IO();
c_ACT_Statistics_Station_1();
d_ACT_Set_Events_Station_1();

ACTION a_ACT_Ctrl_Station_1:
/////////////////////////////////////////////////////////////////////////////////////UTILITIES/////////////////////////////////////////////////////////////////////////////////////
tonStationStopped( IN := bStopped[0] AND bStopped[1], PT := T#1S);
tonExecute(IN := stLeakTesters.State = E_LeakTester_State.RUN_LEAK_TESTERS, PT := T#500MS);
tonWaitResults(IN := (stLeakTesters.State = E_LeakTester_State.WAIT_RESULTS), PT := T#100MS);

/////////////////////////////////////////////////////////////////////////////////////CONDITIONS/////////////////////////////////////////////////////////////////////////////////////

IF stLeakTesters.CMD.bAbort OR bError[0] OR bError[1] THEN
								
	stLeakTesters.State											:= E_LeakTester_State.RESET;
	

END_IF



CASE stLeakTesters.State OF
	
	E_LeakTester_State.ABORTED:
	
								IF stLeakTesters.CMD.bEnable AND NOT bError[0] THEN
									stLeakTesters.State			:= E_LeakTester_State.HOMING;
								ELSIF bError[0] OR bError[1] THEN
									stLeakTesters.State			:= E_LeakTester_State.ERROR;
								END_IF
	
	E_LeakTester_State.HOMING:
	
								IF bReady[0] AND bReady[1] AND bStopped[0] AND bStopped[1] THEN
									stLeakTesters.State			:= E_LeakTester_State.READY;
								
								END_IF
								
	E_LeakTester_State.READY:
	
								IF stLeakTesters.CMD.bExecute THEN
									
									stLeakTesters.State			:= E_LeakTester_State.RUN_LEAK_TESTERS;
								
								END_IF
		
								
	E_LeakTester_State.RUN_LEAK_TESTERS:	
								
								IF stLeakTesters.CMD.LeakTestersCMD.RunLeakTester1 AND stLeakTesters.CMD.LeakTestersCMD.RunLeakTester2 THEN
										
										bStart[0]				:= TRUE;
										bStart[1]				:= TRUE;
									
								ELSIF stLeakTesters.CMD.LeakTestersCMD.RunLeakTester1 AND NOT stLeakTesters.CMD.LeakTestersCMD.RunLeakTester2 THEN
										
										bStart[0]				:= TRUE;
									
								ELSIF NOT stLeakTesters.CMD.LeakTestersCMD.RunLeakTester1 AND stLeakTesters.CMD.LeakTestersCMD.RunLeakTester2 THEN
										
										bStart[1]				:= TRUE;
									
								END_IF
								
								IF tonExecute.Q THEN
									
									stLeakTesters.State			:= E_LeakTester_State.WAIT_LEAK_TESTERS;
								
								END_IF
	
	E_LeakTester_State.WAIT_LEAK_TESTERS:
	
								IF stLeakTesters.CMD.LeakTestersCMD.RunLeakTester1 AND stLeakTesters.CMD.LeakTestersCMD.RunLeakTester2 THEN
										
										IF bLeakTestDone[0] AND bLeakTestDone[1] THEN
											
											stLeakTesters.State	:= E_LeakTester_State.WAIT_RESULTS;
											
										END_IF
									
								ELSIF stLeakTesters.CMD.LeakTestersCMD.RunLeakTester1 AND NOT stLeakTesters.CMD.LeakTestersCMD.RunLeakTester2 THEN
										
										IF bLeakTestDone[0]  THEN
											
											stLeakTesters.State	:= E_LeakTester_State.WAIT_RESULTS;
											
										END_IF
									
								ELSIF NOT stLeakTesters.CMD.LeakTestersCMD.RunLeakTester1 AND stLeakTesters.CMD.LeakTestersCMD.RunLeakTester2 THEN
										
										IF bLeakTestDone[1]  THEN
											
											stLeakTesters.State	:= E_LeakTester_State.WAIT_RESULTS;
											
										END_IF
									
								END_IF
	
	E_LeakTester_State.WAIT_RESULTS:
	
								IF tonWaitResults.Q THEN
									
									stLeakTesters.State	:= E_LeakTester_State.RESULTS;
									
								END_IF


		
	E_LeakTester_State.RESULTS:
								
								IF stLeakTesters.CMD.LeakTestersCMD.RunLeakTester1 THEN
									
									IF bPass[0] THEN
									
										stCycleDataNest1.LeakTest_Pass := TRUE;
										stCycleDataNest1.LeakTest_Fail := FALSE;
										
										stLeakTesters.State	:= E_LeakTester_State.DONE;
								
									ELSIF bFail[0] THEN
									
										stCycleDataNest1.LeakTest_Fail := TRUE;
										stCycleDataNest1.LeakTest_Pass := FALSE;
								
										stLeakTesters.State	:= E_LeakTester_State.DONE;
										
								END_IF
									
								END_IF
								
								IF stLeakTesters.CMD.LeakTestersCMD.RunLeakTester2 THEN
									
									IF bPass[1] THEN
									
										stCycleDataNest2.LeakTest_Pass := TRUE;
										stCycleDataNest2.LeakTest_Fail	:= FALSE;
										
										stLeakTesters.State	:= E_LeakTester_State.DONE;
								
									ELSIF bFail[1] THEN
									
										stCycleDataNest2.LeakTest_Fail	:= TRUE;
										stCycleDataNest2.LeakTest_Pass := FALSE;
										
										stLeakTesters.State	:= E_LeakTester_State.DONE;
								
								END_IF
									
								END_IF
								
								
								
		E_LeakTester_State.DONE:
								IF  stLeakTesters.CMD.bAcknowledge THEN
									
									stLeakTesters.CMD.bAcknowledge := FALSE;
									stLeakTesters.State			:= E_LeakTester_State.RESET;
									
								END_IF	
								
								
								
	E_LeakTester_State.RESET:
	

								bStart[0]						:= FALSE;
								bStart[1]						:= FALSE;
								bReset[0]						:= FALSE;
								bReset[1]						:= FALSE;
								bStop[0]						:= FALSE;
								bStop[1]						:= FALSE;
								bLeakTestDone[0]				:= FALSE;
								bLeakTestDone[1]				:= FALSE;
								bPass[0]						:= FALSE;
								bPass[1]						:= FALSE;
								bFail[0]						:= FALSE;
								bFail[1]						:= FALSE;
								
								IF bError[0] OR bError[1] THEN

									stLeakTesters.State		:= E_LeakTester_State.ERROR;

								ELSIF stLeakTesters.CMD.bAbort OR stLeakTesters.CMD.bEndCycle THEN
									
									stLeakTesters.State			:= E_LeakTester_State.ABORTED;
									
								ELSE stLeakTesters.State			:= E_LeakTester_State.READY;
								
								END_IF
								
								
								
	E_LeakTester_State.STOPPING: 
	
								bStop[0]						:= TRUE;
								bStop[1]						:= TRUE;
								
								IF tonStationStopped.Q THEN
									
									stLeakTesters.State			:= E_LeakTester_State.RESET;
									
								END_IF
	
	E_LeakTester_State.ERROR:
	
								IF NOT bError[0] AND bError[1] THEN
									
									stLeakTesters.State						:= E_LeakTester_State.ABORTED;
									
								END_IF

ELSE stLeakTesters.State := E_LeakTester_State.ABORTED;
	
END_CASE
/////////////////////////////////////////////////////////////////////////////////////STATUS/////////////////////////////////////////////////////////////////////////////////////

stLeakTesters.Status.bBusy	:= 	stLeakTesters.State = E_LeakTester_State.STOPPING OR
								stLeakTesters.State = E_LeakTester_State.HOMING OR
								stLeakTesters.State = E_LeakTester_State.RUN_LEAK_TESTERS OR
								stLeakTesters.State = E_LeakTester_State.WAIT_LEAK_TESTERS;

stLeakTesters.Status.bDone	:= 	stLeakTesters.State = E_LeakTester_State.DONE;

stLeakTesters.Status.bError	:= 	stLeakTesters.State = E_LeakTester_State.ERROR;	

stLeakTesters.Status.bReady	:=	stLeakTesters.State = E_LeakTester_State.READY;

stLeakTesters.Status.bStopped := NOT stLeakTesters.Status.bBusy;
END_ACTION

ACTION b_ACT_IO:


bStopped[0]								:= NOT LeakTester1_IO.sti28General_I_O.bTestActiveLiveData;
bStopped[1]								:= NOT LeakTester2_IO.sti28General_I_O.bTestActiveLiveData;
bError[0]								:= LeakTester1_IO.sti28General_I_O.bMalfunction;
bError[1]								:= LeakTester2_IO.sti28General_I_O.bMalfunction;
bReady[0]								:= LeakTester1_IO.sti28General_I_O.bInstrumentReady;
bReady[1]								:= LeakTester2_IO.sti28General_I_O.bInstrumentReady;
LeakTester1_IO.sti28General_I_O.bReset	:= bReset[0] OR bLeaktester1_Reset;	
LeakTester2_IO.sti28General_I_O.bReset	:= bReset[1] OR bLeaktester2_Reset;	
LeakTester1_IO.sti28General_I_O.bStart	:= bStart[0] OR bLeaktester1_Start;
LeakTester2_IO.sti28General_I_O.bStart	:= bStart[1] OR bLeaktester2_Start;
LeakTester1_IO.sti28General_I_O.bStop	:= bStop[0] OR bLeaktester1_Stop OR stLeakTesters.CMD.bAbort;
LeakTester2_IO.sti28General_I_O.bStop	:= bStop[1] OR bLeaktester2_Stop OR stLeakTesters.CMD.bAbort;



rReset[0](CLK := stLeakTesters.CMD.bReset, Q => bReset[0]);
rReset[1](CLK := stLeakTesters.CMD.bReset, Q => bReset[1]);

fLeakTestDone[0](CLK := LeakTester1_IO.sti28General_I_O.bTestActiveLiveData);
fLeakTestDone[1](CLK := LeakTester2_IO.sti28General_I_O.bTestActiveLiveData);
rPass[0](CLK := LeakTester1_IO.sti28General_I_O.bProgramAccept);
rPass[1](CLK := LeakTester2_IO.sti28General_I_O.bProgramAccept);
rFail[0](CLK := LeakTester1_IO.sti28General_I_O.bProgramReject);
rFail[1](CLK := LeakTester2_IO.sti28General_I_O.bProgramReject);



IF fLeakTestDone[0].Q THEN
	
	bLeakTestDone[0]					:= TRUE;
	
END_IF

IF fLeakTestDone[1].Q THEN
	
	bLeakTestDone[1]					:= TRUE;
	
END_IF

IF rPass[0].Q THEN
	
	bPass[0]							:= TRUE;

END_IF

IF rPass[1].Q THEN
	
	bPass[1]							:= TRUE;

END_IF

IF rFail[0].Q THEN
	
	bFail[0]							:= TRUE;

END_IF

IF rFail[1].Q THEN
	
	bFail[1]							:= TRUE;

END_IF
END_ACTION

ACTION c_ACT_Statistics_Station_1:
stStatisticsHMI[2].sName			:= 'LEAK TESTER 1';
stStatisticsHMI[3].sName			:= 'LEAK TESTER 2';


rGoodStatistics[0]( CLK := stCycleDataNest1.LeakTest_Pass );
rGoodStatistics[1]( CLK := stCycleDataNest2.LeakTest_Pass );
rBadStatistics[0] ( CLK := stCycleDataNest1.LeakTest_Fail );
rBadStatistics[1] ( CLK := stCycleDataNest2.LeakTest_Fail );

IF 	rGoodStatistics[0].Q THEN
	
	stStatisticsHMI[2].nGood		:= stStatisticsHMI[2].nGood + 1;
	
END_IF
								
IF 	rBadStatistics[0].Q THEN
	
	stStatisticsHMI[2].nBad			:= stStatisticsHMI[2].nBad + 1;
	
END_IF

IF stStatisticsHMI[2].bResetGood THEN
	stStatisticsHMI[2].nGood		:= 0;
END_IF

IF stStatisticsHMI[2].bResetBad THEN
	stStatisticsHMI[2].nBad			:= 0;
END_IF


IF 	rGoodStatistics[1].Q THEN
	
	stStatisticsHMI[3].nGood		:= stStatisticsHMI[3].nGood + 1;
	
END_IF
								
IF 	rBadStatistics[1].Q THEN
	
	stStatisticsHMI[3].nBad			:= stStatisticsHMI[3].nBad + 1;
	
END_IF

IF stStatisticsHMI[3].bResetGood THEN
	stStatisticsHMI[3].nGood		:= 0;
END_IF

IF stStatisticsHMI[3].bResetBad THEN
	stStatisticsHMI[3].nBad			:= 0;
END_IF



IF (( stStatisticsHMI[2].nGood + stStatisticsHMI[2].nBad) <> 0) THEN
	
	rEfficency[0]							:= LREAL_TO_FMTSTR(in := (DINT_TO_REAL(stStatisticsHMI[2].nGood) /( DINT_TO_REAL(stStatisticsHMI[2].nGood) + DINT_TO_REAL(stStatisticsHMI[2].nBad))) * 100.0,iPrecision := 2, bRound := TRUE);
	stStatisticsHMI[2].nEfficency		:= CONCAT(STR1 := '%', STR2 := (rEfficency[0]));

ELSE stStatisticsHMI[2].nEfficency		:= CONCAT(STR1 := '%', STR2 := (DINT_TO_STRING(0)));
	
END_IF

IF (( stStatisticsHMI[3].nGood + stStatisticsHMI[3].nBad) <> 0) THEN
	
	rEfficency[1]							:= LREAL_TO_FMTSTR(in := (DINT_TO_REAL(stStatisticsHMI[3].nGood) /( DINT_TO_REAL(stStatisticsHMI[3].nGood) + DINT_TO_REAL(stStatisticsHMI[3].nBad))) * 100.0,iPrecision := 2, bRound := TRUE);
	stStatisticsHMI[3].nEfficency		:= CONCAT(STR1 := '%', STR2 := (rEfficency[1]));

ELSE stStatisticsHMI[3].nEfficency		:= CONCAT(STR1 := '%', STR2 := (DINT_TO_STRING(0)));
	
END_IF
END_ACTION

ACTION d_ACT_Set_Events_Station_1:
//IMMEDIATE FAULTS

stStationEvents[1].aEvents[0].bFault						:= TRUE;
stStationEvents[1].aEvents[0].bEventTimer( IN := (stLeakTesters.State = E_LeakTester_State.RUN_LEAK_TESTERS) OR (stLeakTesters.State = E_LeakTester_State.WAIT_LEAK_TESTERS), PT := stTimers.tStation1TimeOut);
stStationEvents[1].aEvents[0].bEventFlag					:= stStationEvents[1].aEvents[0].bEventTimer.Q;
stStationEvents[1].aEvents[0].bEventText					:= 'Leak tester cycle Timeout';
stStationEvents[1].aEvents[0].sSolution						:= 'Reset System';



//CYCLE STOP REQUEST

stStationEvents[1].aEvents[20].bCycleStopRequest				:= TRUE;
stStationEvents[1].aEvents[20].bEventFlag					:= NOT bReady[0] AND (stLeakTesters.State = E_LeakTester_State.HOMING);// AND (stLeakTesters.State = E_LeakTester_State.HOMING);
stStationEvents[1].aEvents[20].bEventText					:= 'Leak Tester 1 not ready';
stStationEvents[1].aEvents[20].sSolution						:= 'Check Leak tester 1';

stStationEvents[1].aEvents[21].bCycleStopRequest				:= TRUE;
stStationEvents[1].aEvents[21].bEventFlag					:= NOT bReady[1] AND (stLeakTesters.State = E_LeakTester_State.HOMING);// AND (stLeakTesters.State = E_LeakTester_State.HOMING);
stStationEvents[1].aEvents[21].bEventText					:= 'Leak Tester 2 not ready';
stStationEvents[1].aEvents[21].sSolution						:= 'Check Leak tester 2';

stStationEvents[1].aEvents[22].bCycleStopRequest			:= TRUE;
stStationEvents[1].aEvents[22].bEventFlag					:= bError[0] AND bNest1Flag;
stStationEvents[1].aEvents[22].bEventText					:= 'Leak Tester 1 malfunction';
stStationEvents[1].aEvents[22].sSolution					:= 'Check Leak tester 1';

stStationEvents[1].aEvents[23].bCycleStopRequest			:= TRUE;
stStationEvents[1].aEvents[23].bEventFlag					:=  bError[1] AND bNest2Flag;
stStationEvents[1].aEvents[23].bEventText					:= 'Leak Tester 2 malfunction';
stStationEvents[1].aEvents[23].sSolution					:= 'Check Leak tester 2';



//Message
(*
stStationEvents[1].aEvents[3].bMessage						:= TRUE;
stStationEvents[1].aEvents[3].bEventFlag					:= bEventsFlag[3];
stStationEvents[1].aEvents[3].bEventText					:= 'Message 3';
stStationEvents[1].aEvents[3].sSolution						:= '';*)
END_ACTION

END_PROGRAM

// ---- POUs/B_STATIONS/B_3_CAMERA/B_3_1_PRG_Master_Camera.TcPOU
PROGRAM B_3_1_PRG_Master_Camera

VAR
	
	rGoodStatistics						: ARRAY [0..1] OF R_TRIG;
	rBadStatistics						: ARRAY [0..1] OF R_TRIG;
	rEfficency							: ARRAY [0..1] OF STRING(510);
	bEventsFlag							: ARRAY [0..100] OF BOOL;
/////////////////////////////////////////////////////////////////////////////////////I O/////////////////////////////////////////////////////////////////////////////////////	
	bError								: ARRAY [1..4] OF BOOL;
	rReset								: R_TRIG;
	bReset								: BOOL;
	bReady								: BOOL;
	bDone								: ARRAY [1..2] OF BOOL;
	bPass								: ARRAY [1..2] OF BOOL;
	rsPass								: ARRAY [1..2] OF RS;
	bFail								: ARRAY [1..2] OF BOOL;
	bTtigger							: ARRAY [1..4] OF BOOL;
	bTriggerFail						: ARRAY [1..4] OF BOOL;
	bBusy								: ARRAY [1..4] OF BOOL;
	bGeneralBusy						: BOOL;
	bClearBuffer						: BOOL;
	tonTakingPicture					: TON;

	rTriggerCounter						: R_TRIG;
	ctuTriggerCounter					: CTU;
	abReTakingPicture					: ARRAY [1..2] OF BOOL;
	btest								: BOOL;
	rtest								: R_TRIG;
	
	bInspectRequest 					: ARRAY [1..2] OF BOOL; (*Bugfix 03 - 09Jul26 | Code stucks with only one nest enabled*)
	
END_VAR

d_ACT_Set_Events_Station_3();
a_ACT_Ctrl_Station_3();
b_ACT_IO();
c_ACT_Statistics_Station_3();

ACTION a_ACT_Ctrl_Station_3:
/////////////////////////////////////////////////////////////////////////////////////UTILITIES/////////////////////////////////////////////////////////////////////////////////////
tonTakingPicture(PT := T#100MS);
ctuTriggerCounter();
/////////////////////////////////////////////////////////////////////////////////////CONDITIONS/////////////////////////////////////////////////////////////////////////////////////

IF bError[1] OR bError[2] OR bError[3] OR bError[4] OR stCamera.CMD.bAbort THEN
	
	stCamera.State						:= E_Camera_State.RESET_CMD;

END_IF

CASE stCamera.State OF
	
	E_Camera_State.ABORTED:
	
								
								
	
								IF  stCamera.CMD.bEnable THEN
									
									stCamera.State						:= E_Camera_State.HOMING;
								
								END_IF
													
	E_Camera_State.HOMING:
	
								IF bReady THEN
									
									stCamera.State						:= E_Camera_State.READY;
									
								END_IF
	
						
	E_Camera_State.READY:
								bClearBuffer							:= TRUE;
							
								IF stCamera.CMD.bExecute THEN
									
									bInspectRequest[1] := stCamera.CMD.CameraCMD.Inspect1; (*Renan Bugfix 03 - 09Jul26*)
       								bInspectRequest[2] := stCamera.CMD.CameraCMD.Inspect2; (*Renan Bugfix 03 - 09Jul26*)
									
									IF abMachineDefinition[1] THEN
										
										stCamera.State						:= E_Camera_State.TAKING_PICTURE_CAP;
										bClearBuffer						:= FALSE;
										
									ELSIF abMachineDefinition[2] THEN

										stCamera.State						:= E_Camera_State.TAKING_PICTURE_FPB;
										bClearBuffer						:= FALSE;
	
									END_IF
									
								END_IF
	
	E_Camera_State.TAKING_PICTURE_CAP:
								
								bClearBuffer							:= FALSE;
								
								IF bInspectRequest[1] AND bInspectRequest[2] THEN (*Renan Bugfix 03 - 09Jul26*)
																		
									bTtigger[1]							:= TRUE;
									bTtigger[2]							:= TRUE;
									bTtigger[3]							:= TRUE;
									bTtigger[4]							:= TRUE;									
									
									IF bDone[1] AND bDone[2] AND NOT bGeneralBusy  THEN
										
										bTtigger[1]						:= FALSE;
										bTtigger[2]						:= FALSE;
										bTtigger[3]						:= FALSE;
										bTtigger[4]						:= FALSE;
										
										tonTakingPicture.IN				:= TRUE;
								
										IF tonTakingPicture.Q THEN
											
											anCameraScore[1]	:= CONCAT( STR1:= UINT_TO_STRING(Camera1_IO.nScore), STR2 := '%');
											anCameraScore[2]	:= CONCAT( STR1:= UINT_TO_STRING(Camera2_IO.nScore), STR2 := '%');
											anCameraScore[3]	:= CONCAT( STR1:= UINT_TO_STRING(Camera3_IO.nScore), STR2 := '%');
											anCameraScore[4]	:= CONCAT( STR1:= UINT_TO_STRING(Camera4_IO.nScore), STR2 := '%');
											
											stCamera.State						:=	E_Camera_State.COMPARING_RESULTS;
											
										END_IF
										
									END_IF
									
								ELSIF bInspectRequest[1] AND NOT bInspectRequest[2] THEN (*Renan Bugfix 03 - 09Jul26*)
									
									bTtigger[1]							:= TRUE;
									bTtigger[2]							:= TRUE;
									
									IF bDone[1] AND NOT bGeneralBusy THEN
										
										bTtigger[1]						:= FALSE;
										bTtigger[2]						:= FALSE;
									
										tonTakingPicture.IN				:= TRUE;
										
										IF tonTakingPicture.Q THEN
											
											anCameraScore[1]	:= CONCAT( STR1:= UINT_TO_STRING(Camera1_IO.nScore), STR2 := '%');
											anCameraScore[2]	:= CONCAT( STR1:= UINT_TO_STRING(Camera2_IO.nScore), STR2 := '%');
											
											stCamera.State						:=	E_Camera_State.COMPARING_RESULTS;
											
										END_IF
										
									END_IF
								
								ELSIF NOT bInspectRequest[1] AND bInspectRequest[2] THEN (*Renan Bugfix 03 - 09Jul26*)
									
									bTtigger[3]							:= TRUE;
									bTtigger[4]							:= TRUE;
									
									IF bDone[2] AND NOT bGeneralBusy THEN

										bTtigger[3]						:= FALSE;
										bTtigger[4]						:= FALSE;
										
										tonTakingPicture.IN				:= TRUE;
										
										IF tonTakingPicture.Q THEN
											
											anCameraScore[3]	:= CONCAT( STR1:= UINT_TO_STRING(Camera3_IO.nScore), STR2 := '%');
											anCameraScore[4]	:= CONCAT( STR1:= UINT_TO_STRING(Camera4_IO.nScore), STR2 := '%');
											
											stCamera.State						:= 	E_Camera_State.COMPARING_RESULTS;
											
										END_IF
										
										
									END_IF
								
									
								END_IF
								
	E_Camera_State.TAKING_PICTURE_FPB:
	
								bClearBuffer							:= FALSE;
								
								IF stCamera.CMD.CameraCMD.Inspect1 AND stCamera.CMD.CameraCMD.Inspect2 THEN
																		
										bTtigger[1]							:= TRUE;
										bTtigger[2]							:= TRUE;									
									
									IF bDone[1] AND bDone[2] AND NOT bGeneralBusy  THEN
										
										bTtigger[1]						:= FALSE;
										bTtigger[2]						:= FALSE;
										
										tonTakingPicture.IN				:= TRUE;
								
										IF tonTakingPicture.Q THEN
											
											anCameraScore[1]	:= CONCAT( STR1:= UINT_TO_STRING(Camera1_IO.nScore), STR2 := '%');
											anCameraScore[2]	:= CONCAT( STR1:= UINT_TO_STRING(Camera2_IO.nScore), STR2 := '%');
											
											stCamera.State							:= E_Camera_State.COMPARING_RESULTS;
											
										END_IF
										
									END_IF
									
								ELSIF stCamera.CMD.CameraCMD.Inspect1 AND NOT stCamera.CMD.CameraCMD.Inspect2 THEN
									
									bTtigger[1]							:= TRUE;
									
									IF bDone[1] AND NOT bGeneralBusy THEN
										
										bTtigger[1]						:= FALSE;
									
										tonTakingPicture.IN				:= TRUE;
										
										IF tonTakingPicture.Q THEN
											
											anCameraScore[1]	:= CONCAT( STR1:= UINT_TO_STRING(Camera1_IO.nScore), STR2 := '%');
											
											stCamera.State							:= E_Camera_State.COMPARING_RESULTS;
											
										END_IF
										
									END_IF
								
								ELSIF NOT stCamera.CMD.CameraCMD.Inspect1 AND stCamera.CMD.CameraCMD.Inspect2 THEN
									
									bTtigger[2]							:= TRUE;
									
									IF bDone[2] AND NOT bGeneralBusy THEN

										bTtigger[2]						:= FALSE;
										
										tonTakingPicture.IN				:= TRUE;
										
										IF tonTakingPicture.Q THEN
											
											anCameraScore[2]	:= CONCAT( STR1:= UINT_TO_STRING(Camera3_IO.nScore), STR2 := '%');						
											stCamera.State							:= E_Camera_State.COMPARING_RESULTS;
											
										END_IF
										
										
									END_IF
								
									
								END_IF
															
	E_Camera_State.COMPARING_RESULTS:	
	
								tonTakingPicture.IN							:= FALSE;
	
								IF abMachineDefinition[1] THEN
									
									
									ctuTriggerCounter.CU					:= FALSE;
							
									IF stCamera.CMD.CameraCMD.Inspect1 THEN
									
										IF Camera1_IO.bTotalResult = TRUE AND Camera2_IO.bTotalResult = TRUE THEN
										
											bPass[1]							:= TRUE;
											bFail[1]							:= FALSE;
											stCamera.CMD.CameraCMD.Inspect1		:= FALSE;
									
										ELSIF Camera1_IO.bTotalResult = FALSE AND Camera2_IO.bTotalResult = FALSE THEN
										
											bPass[1]							:= FALSE;
											bFail[1]							:= TRUE;
											stCamera.CMD.CameraCMD.Inspect1		:= FALSE;
										
										ELSIF Camera1_IO.bTotalResult <> Camera2_IO.bTotalResult AND ctuTriggerCounter.CV = 5 THEN
										
											bPass[1]							:= FALSE;
											bFail[1]							:= TRUE;
										
										END_IF
								
									END_IF
								
									IF stCamera.CMD.CameraCMD.Inspect2 THEN
									
										IF Camera3_IO.bTotalResult = TRUE AND Camera4_IO.bTotalResult = TRUE THEN
										
											bPass[2]							:= TRUE;
											bFail[2]							:= FALSE;
											stCamera.CMD.CameraCMD.Inspect2		:= FALSE;
									
										ELSIF Camera3_IO.bTotalResult = FALSE AND Camera4_IO.bTotalResult = FALSE THEN
										
											bPass[2]							:= FALSE;
											bFail[2]							:= TRUE;
											stCamera.CMD.CameraCMD.Inspect2		:= FALSE;
										
										ELSIF Camera3_IO.bTotalResult <> Camera4_IO.bTotalResult AND ctuTriggerCounter.CV = 5 THEN
										
											bPass[2]							:= FALSE;
											bFail[2]							:= TRUE;
										
										END_IF
								
									END_IF
									
									stCamera.State								:= E_Camera_State.RESULTS_CAP;
								
								ELSIF abMachineDefinition[2] THEN

									IF stCamera.CMD.CameraCMD.Inspect1 THEN
										
										IF Camera1_IO.bTotalResult THEN
										
											bPass[1]							:= TRUE;
											bFail[1]							:= FALSE;
											stCamera.CMD.CameraCMD.Inspect1		:= FALSE;
									
										ELSE 
											bPass[1]							:= FALSE;
											bFail[1]							:= TRUE;
											stCamera.CMD.CameraCMD.Inspect1		:= FALSE;
											
										END_IF
																		
									END_IF

								
									IF stCamera.CMD.CameraCMD.Inspect2 THEN
										
										IF Camera2_IO.bTotalResult THEN
										
											bPass[2]							:= TRUE;
											bFail[2]							:= FALSE;
											stCamera.CMD.CameraCMD.Inspect2		:= FALSE;
									
										ELSE 
											bPass[2]							:= FALSE;
											bFail[2]							:= TRUE;
											stCamera.CMD.CameraCMD.Inspect2		:= FALSE;
										
										
										END_IF
										
										
										
									END_IF
										
									stCamera.State								:= E_Camera_State.RESULTS_FPB;
									
								END_IF
				
								
								
								
								
		E_Camera_State.RESULTS_CAP: (*Renan Bugfix 03 - 09Jul26 | Entire case*)

								IF ((bPass[1] OR bFail[1]) OR NOT bInspectRequest[1]) AND
								   ((bPass[2] OR bFail[2]) OR NOT bInspectRequest[2]) THEN
							
									IF bInspectRequest[1] THEN
										stCycleDataNest1.Camera_Pass := bPass[1];
										stCycleDataNest1.Camera_Fail := bFail[1];
									END_IF
							
									IF bInspectRequest[2] THEN
										stCycleDataNest2.Camera_Pass := bPass[2];
										stCycleDataNest2.Camera_Fail := bFail[2];
									END_IF
							
									stCamera.State := E_Camera_State.DONE;
									ctuTriggerCounter.RESET := TRUE;
							
								ELSE
							
									ctuTriggerCounter.CU := TRUE;
							
									bTtigger[1] := FALSE;
									bTtigger[2] := FALSE;
									bTtigger[3] := FALSE;
									bTtigger[4] := FALSE;
							
									bClearBuffer := TRUE;
							
									stCamera.State := E_Camera_State.TAKING_PICTURE_CAP;
							
								END_IF

		E_Camera_State.RESULTS_FPB:			
		
								
								stCycleDataNest1.Camera_Pass			:= bPass[1];
								stCycleDataNest1.Camera_Fail			:= bFail[1];
								stCycleDataNest2.Camera_Pass			:= bPass[2];
								stCycleDataNest2.Camera_Fail			:= bFail[2];
								
								stCamera.State							:= E_Camera_State.DONE;
								
		E_Camera_State.DONE:		
	
								IF stCamera.CMD.bAcknowledge THEN
									
									stCamera.CMD.bAcknowledge			:= FALSE;
									stCamera.State						:= E_Camera_State.RESET_CMD;
								
								END_IF
								
	E_Camera_State.RESET_CMD:						
	
								
									
								bTtigger[1]								:= FALSE;
								bTtigger[2]								:= FALSE;
								bTtigger[3]								:= FALSE;
								bTtigger[4]								:= FALSE;
								
								bPass[1]								:= FALSE;
								bPass[2]								:= FALSE;
								bFail[1]								:= FALSE;
								bFail[2]								:= FALSE;
								ctuTriggerCounter.RESET					:= FALSE;
								ctuTriggerCounter.CU					:= FALSE;
								
								bInspectRequest[1] 						:= FALSE; (*Renan Bugfix 03 - 09Jul26*)
								bInspectRequest[2] 						:= FALSE; (*Renan Bugfix 03 - 09Jul26*)
					
								IF  bError[1] OR bError[2] OR bError[3] OR bError[4] THEN
									
									stCamera.State						:= E_Camera_State.ERROR;
									
								ELSIF  stCamera.CMD.bAbort THEN

									stCamera.State						:= E_Camera_State.ABORTED;
								
								ELSE 
									stCamera.State						:= E_Camera_State.READY;
								END_IF
								
								

								
	
	E_Camera_State.ERROR:	
	
								IF NOT bError[1] OR bError[2] OR bError[3] OR bError[4] THEN
									
									stCamera.State					:= E_Camera_State.ABORTED;
								
								END_IF
					
								
									

ELSE stCamera.State						:= E_Camera_State.READY;
	
END_CASE
/////////////////////////////////////////////////////////////////////////////////////STATUS/////////////////////////////////////////////////////////////////////////////////////

stCamera.Status.bBusy		:= 	(stCamera.State	= E_Camera_State.TAKING_PICTURE_CAP) OR (stCamera.State	= E_Camera_State.TAKING_PICTURE_FPB);
								
stCamera.Status.bDone		:=	stCamera.State	= E_Camera_State.DONE;
											
stCamera.Status.bError		:= 	stCamera.State	= E_Camera_State.ERROR;

stCamera.Status.bReady		:= 	stCamera.State	= E_Camera_State.READY;

stCamera.Status.bStopped	:= 	NOT stCamera.Status.bBusy;
END_ACTION

ACTION b_ACT_IO:


bError[1]								:= Camera1_IO.bError;
bError[2]								:= Camera2_IO.bError;
bError[3]								:= Camera3_IO.bError;
bError[4]								:= Camera4_IO.bError;

IF abMachineDefinition[1] THEN
	
	bReady								:=  (Camera1_IO.bReady AND Camera1_IO.bRun) AND (Camera2_IO.bReady AND Camera2_IO.bRun) AND 
											(Camera3_IO.bReady AND Camera3_IO.bRun) AND (Camera4_IO.bReady AND Camera4_IO.bRun);
											
	bDone[1]							:= Camera1_IO.bResultReady AND Camera2_IO.bResultReady;
	bDone[2]							:= Camera3_IO.bResultReady AND Camera4_IO.bResultReady;
											
	rsPass[1]( SET := bDone[1] AND (Camera1_IO.bTotalResult = TRUE AND Camera2_IO.bTotalResult = TRUE), RESET1 := (stCamera.State = E_Camera_State.ABORTED) OR (stCamera.State = E_Camera_State.READY));
	rsPass[2]( SET := bDone[2] AND (Camera3_IO.bTotalResult = TRUE AND Camera4_IO.bTotalResult = TRUE), RESET1 := (stCamera.State = E_Camera_State.ABORTED) OR (stCamera.State = E_Camera_State.READY));
	
	bGeneralBusy						:= bBusy[1] OR bBusy[2] OR bBusy[3] OR bBusy[4];

ELSIF abMachineDefinition[2] THEN
	
	bReady								:=  (Camera1_IO.bReady AND Camera1_IO.bRun) AND (Camera2_IO.bReady AND Camera2_IO.bRun);
	
	bDone[1]							:= Camera1_IO.bResultReady;
	bDone[2]							:= Camera2_IO.bResultReady;
	
	rsPass[1]( SET := bDone[1] AND Camera1_IO.bTotalResult = TRUE , RESET1 := (stCamera.State = E_Camera_State.ABORTED) OR (stCamera.State = E_Camera_State.READY));
	rsPass[2]( SET := bDone[2] AND Camera2_IO.bTotalResult = TRUE , RESET1 := (stCamera.State = E_Camera_State.ABORTED) OR (stCamera.State = E_Camera_State.READY));

	bGeneralBusy						:= bBusy[1] OR bBusy[2];

END_IF

bBusy[1]								:= Camera1_IO.bBusy;
bBusy[2]								:= Camera2_IO.bBusy;
bBusy[3]								:= Camera3_IO.bBusy;
bBusy[4]								:= Camera4_IO.bBusy;

bTriggerFail[1]							:= Camera1_IO.bTriggerFail;
bTriggerFail[2]							:= Camera2_IO.bTriggerFail;
bTriggerFail[3]							:= Camera3_IO.bTriggerFail;
bTriggerFail[4]							:= Camera4_IO.bTriggerFail;

Camera1_IO.bReset						:= bReset;
Camera2_IO.bReset						:= bReset;
Camera3_IO.bReset						:= bReset;
Camera4_IO.bReset						:= bReset;

Camera1_IO.bTrigger						:= bTtigger[1] OR bCameraTrigger[1];	
Camera2_IO.bTrigger						:= bTtigger[2] OR bCameraTrigger[2];
Camera3_IO.bTrigger						:= bTtigger[3] OR bCameraTrigger[3];
Camera4_IO.bTrigger						:= bTtigger[4] OR bCameraTrigger[4];

IF bClearBuffer	THEN
	
	Camera1_IO.bClearBuffer				:= TRUE;
	Camera2_IO.bClearBuffer				:= TRUE;
	Camera3_IO.bClearBuffer				:= TRUE;
	Camera4_IO.bClearBuffer				:= TRUE;

ELSE

	Camera1_IO.bClearBuffer				:= FALSE;
	Camera2_IO.bClearBuffer				:= FALSE;
	Camera3_IO.bClearBuffer				:= FALSE;
	Camera4_IO.bClearBuffer				:= FALSE;

END_IF

//////////////////////////////////////////////////////////////////////HMI//////////////////////////////////////////////////////////////////////////////
bCameraSettingNo[1]						:= 2;
bCameraSettingNo[2]						:= 2;
bCameraSettingNo[3]						:= 2;
bCameraSettingNo[4]						:= 2;


Camera1_IO.bResetStatistics				:= bCameraResetStatistics[1];
Camera1_IO.bSettingNo					:= bCameraSettingNo[1];
Camera1_IO.bSettingVal					:= bCameraSettingVal[1];
Camera1_IO.bSetTreshold					:= bCameraSetTreshold[1];

Camera2_IO.bResetStatistics				:= bCameraResetStatistics[2];
Camera2_IO.bSettingNo					:= bCameraSettingNo[2];
Camera2_IO.bSettingVal					:= bCameraSettingVal[2];
Camera2_IO.bSetTreshold					:= bCameraSetTreshold[2];

Camera3_IO.bResetStatistics				:= bCameraResetStatistics[3];
Camera3_IO.bSettingNo					:= bCameraSettingNo[3];
Camera3_IO.bSettingVal					:= bCameraSettingVal[3];
Camera3_IO.bSetTreshold					:= bCameraSetTreshold[3];

Camera4_IO.bResetStatistics				:= bCameraResetStatistics[4];
Camera4_IO.bSettingNo					:= bCameraSettingNo[4];
Camera4_IO.bSettingVal					:= bCameraSettingVal[4];
Camera4_IO.bSetTreshold					:= bCameraSetTreshold[4];

//Camera1_IO.bTriggerFail

rReset( CLK := stCamera.CMD.bReset, Q => bReset);
END_ACTION

ACTION c_ACT_Statistics_Station_3:
stStatisticsHMI[6].sName			:= 'Vision System 1';
stStatisticsHMI[7].sName			:= 'Vision System 2';


rGoodStatistics[0]( CLK := stCycleDataNest1.Camera_Pass);
rBadStatistics[0]( CLK := stCycleDataNest1.Camera_Fail);
rGoodStatistics[1]( CLK := stCycleDataNest2.Camera_Pass);
rBadStatistics[1]( CLK := stCycleDataNest2.Camera_Fail);

IF 	rGoodStatistics[0].Q THEN
	
	stStatisticsHMI[6].nGood		:= stStatisticsHMI[6].nGood + 1;
	
END_IF
								
IF 	rBadStatistics[0].Q THEN
	
	stStatisticsHMI[6].nBad			:= stStatisticsHMI[6].nBad + 1;
	
END_IF

IF stStatisticsHMI[6].bResetGood THEN
	stStatisticsHMI[6].nGood		:= 0;
END_IF

IF stStatisticsHMI[6].bResetBad THEN
	stStatisticsHMI[6].nBad			:= 0;
END_IF

IF 	rGoodStatistics[1].Q THEN
	
	stStatisticsHMI[7].nGood		:= stStatisticsHMI[7].nGood + 1;
	
END_IF
								
IF 	rBadStatistics[1].Q THEN
	
	stStatisticsHMI[7].nBad			:= stStatisticsHMI[7].nBad + 1;
	
END_IF

IF stStatisticsHMI[7].bResetGood THEN
	stStatisticsHMI[7].nGood		:= 0;
END_IF

IF stStatisticsHMI[7].bResetBad THEN
	stStatisticsHMI[7].nBad			:= 0;
END_IF

IF (( stStatisticsHMI[6].nGood + stStatisticsHMI[6].nBad) <> 0) THEN
	
	rEfficency[0]							:= LREAL_TO_FMTSTR(in := (DINT_TO_REAL(stStatisticsHMI[6].nGood) /( DINT_TO_REAL(stStatisticsHMI[6].nGood) + DINT_TO_REAL(stStatisticsHMI[6].nBad))) * 100.0,iPrecision := 2, bRound := TRUE);
	stStatisticsHMI[6].nEfficency		:= CONCAT(STR1 := '%', STR2 := (rEfficency[0]));

ELSE stStatisticsHMI[6].nEfficency		:= CONCAT(STR1 := '%', STR2 := (DINT_TO_STRING(0)));
	
END_IF

IF (( stStatisticsHMI[7].nGood + stStatisticsHMI[7].nBad) <> 0) THEN
	
	rEfficency[1]							:= LREAL_TO_FMTSTR(in := (DINT_TO_REAL(stStatisticsHMI[7].nGood) /( DINT_TO_REAL(stStatisticsHMI[7].nGood) + DINT_TO_REAL(stStatisticsHMI[7].nBad))) * 100.0,iPrecision := 2, bRound := TRUE);
	stStatisticsHMI[7].nEfficency		:= CONCAT(STR1 := '%', STR2 := (rEfficency[1]));

ELSE stStatisticsHMI[7].nEfficency		:= CONCAT(STR1 := '%', STR2 := (DINT_TO_STRING(0)));
	
END_IF
END_ACTION

ACTION d_ACT_Set_Events_Station_3:
//IMMEDIATE FAULTS

stStationEvents[3].aEvents[0].bFault						:= TRUE;
stStationEvents[3].aEvents[0].bEventFlag					:= bError[1];
stStationEvents[3].aEvents[0].bEventText					:= 'Error camera 1';
stStationEvents[3].aEvents[0].sSolution						:= 'Check camera 1';

stStationEvents[3].aEvents[1].bFault						:= TRUE;
stStationEvents[3].aEvents[1].bEventFlag					:= bError[2];
stStationEvents[3].aEvents[1].bEventText					:= 'Error camera 2';
stStationEvents[3].aEvents[1].sSolution						:= 'Check camera 2';

stStationEvents[3].aEvents[2].bFault						:= TRUE;
stStationEvents[3].aEvents[2].bEventFlag					:= bError[3];
stStationEvents[3].aEvents[2].bEventText					:= 'Error camera 3';
stStationEvents[3].aEvents[2].sSolution						:= 'Check camera 3';

stStationEvents[3].aEvents[3].bFault						:= TRUE;
stStationEvents[3].aEvents[3].bEventFlag					:= bError[4];
stStationEvents[3].aEvents[3].bEventText					:= 'Error camera 4';
stStationEvents[3].aEvents[3].sSolution						:= 'Check camera 4';

stStationEvents[3].aEvents[4].bFault						:= TRUE;
stStationEvents[3].aEvents[4].bEventTimer(IN := stCamera.Status.bBusy, PT := stTimers.tStation3TimeOut);
stStationEvents[3].aEvents[4].bEventFlag					:= stStationEvents[3].aEvents[4].bEventTimer.Q;
stStationEvents[3].aEvents[4].bEventText					:= 'Camera Cycle Timeout';
stStationEvents[3].aEvents[4].sSolution						:= 'Reset Sytem';


//CYCLE STOP FAULT

stStationEvents[3].aEvents[20].bCycleStopRequest			:= TRUE;
stStationEvents[3].aEvents[20].bEventFlag					:= bTriggerFail[1];
stStationEvents[3].aEvents[20].bEventText					:= 'Trigger failed in camera 1';
stStationEvents[3].aEvents[20].sSolution					:= 'Check camera 1';

stStationEvents[3].aEvents[21].bCycleStopRequest			:= TRUE;
stStationEvents[3].aEvents[21].bEventFlag					:= bTriggerFail[2];
stStationEvents[3].aEvents[21].bEventText					:= 'Trigger failed in camera 2';
stStationEvents[3].aEvents[21].sSolution					:= 'Check camera 2';

stStationEvents[3].aEvents[22].bCycleStopRequest			:= TRUE;
stStationEvents[3].aEvents[22].bEventFlag					:= bTriggerFail[3];
stStationEvents[3].aEvents[22].bEventText					:= 'Trigger failed in camera 3';
stStationEvents[3].aEvents[22].sSolution					:= 'Check camera 3';

stStationEvents[3].aEvents[23].bCycleStopRequest			:= TRUE;
stStationEvents[3].aEvents[23].bEventFlag					:= bTriggerFail[4];
stStationEvents[3].aEvents[23].bEventText					:= 'Trigger failed in camera 4';
stStationEvents[3].aEvents[23].sSolution					:= 'Check camera 4';

stStationEvents[3].aEvents[24].bCycleStopRequest			:= TRUE;
stStationEvents[3].aEvents[24].bEventFlag					:= NOT Camera1_IO.bRun;
stStationEvents[3].aEvents[24].bEventText					:= 'Camera 1 is not in Run mode';
stStationEvents[3].aEvents[24].sSolution					:= 'Go to software and activate Run';

stStationEvents[3].aEvents[25].bCycleStopRequest			:= TRUE;
stStationEvents[3].aEvents[25].bEventFlag					:= NOT Camera2_IO.bRun;
stStationEvents[3].aEvents[25].bEventText					:= 'Camera 2 is not in Run mode';
stStationEvents[3].aEvents[25].sSolution					:= 'Go to software and activate Run';

stStationEvents[3].aEvents[26].bCycleStopRequest			:= TRUE;
stStationEvents[3].aEvents[26].bEventFlag					:= NOT Camera3_IO.bRun AND NOT abMachineDefinition[2];
stStationEvents[3].aEvents[26].bEventText					:= 'Camera 3 is not in Run mode';
stStationEvents[3].aEvents[26].sSolution					:= 'Go to software and activate Run';

stStationEvents[3].aEvents[27].bCycleStopRequest			:= TRUE;
stStationEvents[3].aEvents[27].bEventFlag					:= NOT Camera4_IO.bRun AND NOT abMachineDefinition[2];
stStationEvents[3].aEvents[27].bEventText					:= 'Camera 4 is not in Run mode';
stStationEvents[3].aEvents[27].sSolution					:= 'Go to software and activate Run';
END_ACTION

END_PROGRAM

// ---- POUs/B_STATIONS/B_4_PROCESS_CYLINDER__SLIDE_DOOR/B_4_1_PRG_Master_ProcessCylinder.TcPOU
PROGRAM B_4_1_PRG_Master_ProcessCylinder

VAR

	
	
/////////////////////////////////////////////////////////////////////////////////////I O/////////////////////////////////////////////////////////////////////////////////////	
	bExtended							: BOOL;
	bRetracted							: BOOL;
	bExtend								: BOOL;
	bRetract							: BOOL;

	bProcessDoorClosed					: BOOL;
	
END_VAR

d_ACT_Set_Events_Station_4A();
a_ACT_Ctrl_Station_4A();
b_ACT_IO_A();
c_Manual();

ACTION a_ACT_Ctrl_Station_4A:
/////////////////////////////////////////////////////////////////////////////////////UTILITIES/////////////////////////////////////////////////////////////////////////////////////

/////////////////////////////////////////////////////////////////////////////////////CONDITIONS/////////////////////////////////////////////////////////////////////////////////////


IF stProcessCylinder.CMD.bAbort THEN
	
	stProcessCylinder.State				:= E_ProcessCylinder_State.RESET;

END_IF

CASE stProcessCylinder.State OF
	
	E_ProcessCylinder_State.ABORTED:
	
								IF stProcessCylinder.CMD.bEnable THEN
									
									stProcessCylinder.State				:= E_ProcessCylinder_State.HOMING;
								
								END_IF
								
	E_ProcessCylinder_State.HOMING:
	
								IF bProcessDoorClosed THEN
									
									bRetract							:= TRUE;
									
								END_IF
								
								IF bRetracted THEN
									
									bRetract							:= FALSE;
									stProcessCylinder.State				:= E_ProcessCylinder_State.READY;
									
								
								END_IF
	
	E_ProcessCylinder_State.READY:
	
								IF stProcessCylinder.CMD.bExecute AND stProcessCylinder.CMD.ProcessCylinderCMD.ExtendCylinder1 THEN

									stProcessCylinder.State				:= E_ProcessCylinder_State.EXTEND;
									
								ELSIF stProcessCylinder.CMD.bExecute AND stProcessCylinder.CMD.ProcessCylinderCMD.RetractCylinder1 THEN
									
									stProcessCylinder.State				:= E_ProcessCylinder_State.RETRACT;;									
																		
								END_IF
	
	E_ProcessCylinder_State.EXTEND:
	
								bExtend									:= stProcessCylinder.CMD.ProcessCylinderCMD.ExtendCylinder1;
								
								IF bExtend THEN
									
									IF bExtended THEN

										stProcessCylinder.State			:= E_ProcessCylinder_State.DONE;
									
									END_IF						
	
								END_IF
								
	E_ProcessCylinder_State.RETRACT:
	
								bRetract								:= stProcessCylinder.CMD.ProcessCylinderCMD.RetractCylinder1;
								
								
								IF bRetract THEN
									
									IF bRetracted THEN

										stProcessCylinder.State				:= E_ProcessCylinder_State.DONE;
									
									END_IF					
	
								END_IF
								
	E_ProcessCylinder_State.DONE:
	
								IF stProcessCylinder.CMD.bAcknowledge THEN
									
									stProcessCylinder.CMD.bAcknowledge		:= FALSE;
									stProcessCylinder.State					:= E_ProcessCylinder_State.RESET;
								
								END_IF
	
	
	E_ProcessCylinder_State.RESET:	
	
								bExtend										:= FALSE;								
								bRetract									:= FALSE;
								
								
								IF NOT stProcessCylinder.CMD.bAbort AND NOT stProcessCylinder.CMD.bEndCycle THEN
									
									stProcessCylinder.State					:= E_ProcessCylinder_State.READY;
									
								ELSE stProcessCylinder.State					:= E_ProcessCylinder_State.ABORTED;
								END_IF
									

ELSE stProcessCylinder.State	:= E_ProcessCylinder_State.ABORTED;
	
END_CASE
/////////////////////////////////////////////////////////////////////////////////////STATUS/////////////////////////////////////////////////////////////////////////////////////

stProcessCylinder.Status.bBusy		:= 	stProcessCylinder.State	= E_ProcessCylinder_State.EXTEND OR
										stProcessCylinder.State	= E_ProcessCylinder_State.RETRACT OR 
										stProcessCylinder.State	= E_ProcessCylinder_State.STOPPING;
								
stProcessCylinder.Status.bDone		:=	stProcessCylinder.State	= E_ProcessCylinder_State.DONE;

stProcessCylinder.Status.bReady		:= 	stProcessCylinder.State	= E_ProcessCylinder_State.READY;

stProcessCylinder.Status.bStopped	:= 	NOT stProcessCylinder.Status.bBusy;
END_ACTION

ACTION b_ACT_IO_A:

bExtended								:= dw_T08_EL1809.iProcessCylinderExtended;
bRetracted								:= stTwinSAFE.qProcessCylinderRetracted;

IF bExtend OR bProcessCylinder_Down2 THEN
	
	dw_T09_EL2809.qExtendProcessCylinder	:= TRUE ;
	dw_T09_EL2809.qRetractProcessCylinder	:= FALSE;

ELSIF bRetract OR bProcessCylinder_Up THEN
	
	dw_T09_EL2809.qExtendProcessCylinder	:= FALSE;
	dw_T09_EL2809.qRetractProcessCylinder	:= TRUE;

ELSIF stMachineStatus.bFault THEN
	
	dw_T09_EL2809.qExtendProcessCylinder	:= FALSE;
	dw_T09_EL2809.qRetractProcessCylinder	:= FALSE;

END_IF


IF stStationEvents[3].aEvents[0].bEventTimer.Q THEN
	
	bRetract := FALSE;

END_IF

IF stStationEvents[3].aEvents[1].bEventTimer.Q THEN
	
	bExtended := FALSE;

END_IF

bProcessDoorClosed := dw_T05_EL1918.iProcessDoorClosed1 AND dw_T05_EL1918.iProcessDoorClosed2 AND dw_T05_EL1918.iProcessDoorFB;
END_ACTION

ACTION c_Manual:
(*
IF bProcessCylinder1_Up THEN
	
	bRetract[0] := TRUE;
	
ELSIF bRetracted[0] THEN
	
	bRetract[0] := FALSE;

END_IF

IF bProcessCylinder1_Down THEN
	
	bExtend[0] := TRUE;
	
ELSIF bExtended[0] THEN
	
	bExtend[0] := FALSE;

END_IF

IF bProcessCylinder2_Up THEN
	
	bRetract[1] := TRUE;
	
ELSIF bRetracted[1] THEN
	
	bRetract[1] := FALSE;

END_IF

IF bProcessCylinder2_Down THEN
	
	bExtend[1] := TRUE;
	
ELSIF bExtended[1] THEN
	
	bExtend[1] := FALSE;

END_IF
*)
END_ACTION

ACTION d_ACT_Set_Events_Station_4A:
//FAULTS

stStationEvents[3].aEvents[0].bEventTimer( IN := (bExtend AND NOT bExtended), PT := T#10S);
stStationEvents[3].aEvents[0].bFault						:= TRUE;
stStationEvents[3].aEvents[0].bEventFlag					:= stStationEvents[3].aEvents[0].bEventTimer.Q;
stStationEvents[3].aEvents[0].bEventText					:= 'Process Cylinder 1 extend timeout';
stStationEvents[3].aEvents[0].sSolution						:= 'Check cylinder, neumatic connections and sensors';

stStationEvents[3].aEvents[1].bEventTimer( IN := (bRetract AND NOT bRetracted), PT := T#3S);
stStationEvents[3].aEvents[1].bFault						:= TRUE;
stStationEvents[3].aEvents[1].bEventFlag					:= stStationEvents[3].aEvents[1].bEventTimer.Q;
stStationEvents[3].aEvents[1].bEventText					:= 'Process Cylinder retract timeout';
stStationEvents[3].aEvents[1].sSolution						:= 'Check cylinder, neumatic connections and sensors';


//CYCLE STOP REQUEST

(*stStationEvents[3].aEvents[2].bCycleStopRequest			:= TRUE;
stStationEvents[3].aEvents[2].bEventFlag					:= ;
stStationEvents[3].aEvents[2].bEventText					:= 'ST1 EVENT 7';*)
END_ACTION

END_PROGRAM

// ---- POUs/B_STATIONS/B_4_PROCESS_CYLINDER__SLIDE_DOOR/B_4_2_PRG_Master_ProcessDoor.TcPOU
PROGRAM B_4_2_PRG_Master_ProcessDoor

VAR

	bEventsFlag							: ARRAY [0..100] OF BOOL;
/////////////////////////////////////////////////////////////////////////////////////I O/////////////////////////////////////////////////////////////////////////////////////	
	
	bOpenDoor							: BOOL;
	bCloseDoor							: BOOL;
	bCloseDoorHMI						: BOOL;
	bOpenDoorHMI						: BOOL;
	bDoorClosed							: BOOL;
	tonDoorOpened						: TON;
	bDoorOpened							: BOOL;
	
	bProcessCylinderNotHomed			: BOOL;
	

	
	
END_VAR

d_ACT_Set_Events_Station_4B();
a_ACT_Ctrl_Station_4B();
b_ACT_IO_B();
c_Manual();

ACTION a_ACT_Ctrl_Station_4B:
/////////////////////////////////////////////////////////////////////////////////////UTILITIES/////////////////////////////////////////////////////////////////////////////////////

/////////////////////////////////////////////////////////////////////////////////////CONDITIONS/////////////////////////////////////////////////////////////////////////////////////
IF stProcessDoor.State <> E_ProcessDoor_State.HOMING THEN
	
	bDoorClosingInitFlag											:= FALSE;

END_IF



IF stProcessDoor.CMD.bAbort THEN
	
	stProcessDoor.State				:= E_ProcessDoor_State.RESET;
	
ELSIF stProcessDoor.CMD.bEndCycle THEN
	
	stProcessDoor.State				:= E_ProcessDoor_State.STOPPING;

END_IF

CASE stProcessDoor.State OF
	
	E_ProcessDoor_State.ABORTED:
	
								IF stProcessDoor.CMD.bEnable THEN
									
									stProcessDoor.State				:= E_ProcessDoor_State.HOMING;
								
								END_IF
								
	E_ProcessDoor_State.HOMING: 
	
	
								IF bProcessCylinderNotHomed  THEN
									
									bCloseDoor						:= TRUE; 
									bOpenDoor						:= FALSE;
									
									IF NOT bDoorClosed AND bCloseDoor THEN
										
										bDoorClosingInitFlag		:= TRUE;
									ELSE bDoorClosingInitFlag		:= FALSE;
									END_IF
									
								ELSE
									
									bCloseDoor						:= FALSE;
									bOpenDoor						:= TRUE;
									
								END_IF
								
								IF bDoorOpened AND NOT bProcessCylinderNotHomed THEN
									
									stProcessDoor.State				:= E_ProcessDoor_State.READY;									
									bOpenDoor						:= FALSE;
																	
								END_IF
	
	
	E_ProcessDoor_State.READY:
	
								IF stProcessDoor.CMD.bExecute AND 	stProcessDoor.CMD.ProcessDoorCMD.OpenDoor	THEN

									stProcessDoor.State				:= E_ProcessDoor_State.OPEN;
									
								ELSIF stProcessDoor.CMD.bExecute AND 	stProcessDoor.CMD.ProcessDoorCMD.CloseDoor	THEN
									
									stProcessDoor.State				:= E_ProcessDoor_State.CLOSE;									
																		
								END_IF
	

	E_ProcessDoor_State.OPEN:
	
								bOpenDoor							:= TRUE;
								
								IF bDoorOpened	THEN
									
									stProcessDoor.State				:= E_ProcessDoor_State.DONE;
								
								END_IF
								
	E_ProcessDoor_State.CLOSE:
	
								bCloseDoor							:= TRUE; //Thays
								
								IF bDoorClosed THEN
									
									stProcessDoor.State				:= E_ProcessDoor_State.DONE;
								
								END_IF
								
	E_ProcessDoor_State.DONE:
	
	
								IF stProcessDoor.CMD.bAcknowledge THEN
									
									stProcessDoor.CMD.bAcknowledge	:= FALSE;
									stProcessDoor.State				:= E_ProcessDoor_State.RESET;
								
								END_IF
	
	
	E_ProcessDoor_State.RESET:	
	
								bOpenDoor							:= FALSE;
								bCloseDoor							:= FALSE;
								
								IF NOT stProcessDoor.CMD.bAbort AND NOT stProcessDoor.CMD.bEndCycle THEN
									
									stProcessDoor.State				:= E_ProcessDoor_State.READY;
									
								ELSE stProcessDoor.State			:= E_ProcessDoor_State.ABORTED;
								END_IF
	
					
	E_ProcessDoor_State.STOPPING:					
									
								bOpenDoor							:= TRUE;
									
								IF bDoorOpened THEN
									
									bOpenDoor						:= FALSE;
									stProcessDoor.State				:= E_ProcessDoor_State.RESET;
								
								END_IF
								
							
														
									

ELSE stProcessDoor.State		:= E_ProcessDoor_State.ABORTED;
	
END_CASE
/////////////////////////////////////////////////////////////////////////////////////STATUS/////////////////////////////////////////////////////////////////////////////////////

stProcessDoor.Status.bBusy			:= 	stProcessDoor.State	= E_ProcessDoor_State.CLOSE OR
										stProcessDoor.State	= E_ProcessDoor_State.OPEN OR 
										stProcessDoor.State	= E_ProcessDoor_State.STOPPING;
								
stProcessDoor.Status.bDone			:=	stProcessDoor.State	= E_ProcessDoor_State.DONE;

stProcessDoor.Status.bReady			:= 	stProcessDoor.State	= E_ProcessDoor_State.READY;

stProcessDoor.Status.bStopped		:= 	NOT stProcessDoor.Status.bBusy;
END_ACTION

ACTION b_ACT_IO_B:
tonDoorOpened( IN := NOT bDoorClosed, PT := stTimers.tDoorOpenedSignal);


bDoorClosed								:= dw_T05_EL1918.iProcessDoorClosed1 AND dw_T05_EL1918.iProcessDoorClosed2 AND dw_T05_EL1918.iProcessDoorFB;
bDoorOpened								:= tonDoorOpened.Q; 
bProcessDoorClosed						:= bDoorClosed;


bDoorOpenedFlag							:= bDoorOpened;

dw_T09_EL2809.qOpenProcessDoor	:= bOpenDoor OR bOpenDoorHMI OR stStationEvents[4].aEvents[0].bEventTimer.Q;;	
dw_T09_EL2809.qCloseProcessDoor	:= bCloseDoor OR bCloseDoorHMI;

bProcessCylinderNotHomed				:= NOT stTwinSAFE.qProcessCylinderRetracted;
END_ACTION

ACTION c_Manual:


IF bProcessDoor_Down AND stTwinSAFE.qTwoHandsSafe THEN
	
	bCloseDoorHMI					:= TRUE; 
	bProcessDoor_Down				:= FALSE;
	
ELSIF bDoorClosed  OR NOT stMachineStatus.bManualMode THEN

	 bCloseDoorHMI					:= FALSE;
	 bProcessDoor_Down				:= FALSE;

END_IF

IF bProcessDoor_UP THEN
	
	bOpenDoorHMI					:= TRUE;
	
	
ELSIF bDoorOpened OR  NOT stMachineStatus.bManualMode THEN

	bOpenDoorHMI					:= FALSE;	 
	
END_IF
END_ACTION

ACTION d_ACT_Set_Events_Station_4B:
//IMMEDIATE FAULTS

stStationEvents[4].aEvents[0].bEventTimer( IN :=  (bCloseDoor OR bCloseDoorHMI) AND NOT bDoorClosed, PT := T#2S);
stStationEvents[4].aEvents[0].bFault						:= TRUE;
stStationEvents[4].aEvents[0].bEventFlag					:= stStationEvents[4].aEvents[0].bEventTimer.Q;
stStationEvents[4].aEvents[0].bEventText					:= 'Process Door extend timeout';
stStationEvents[4].aEvents[0].sSolution						:= 'Check cylinder, neumatic connections and sensors';

stStationEvents[4].aEvents[1].bEventTimer( IN :=  (bOpenDoor OR bOpenDoorHMI) AND NOT bDoorOpened, PT := T#2S);
stStationEvents[4].aEvents[1].bFault						:= TRUE;
stStationEvents[4].aEvents[1].bEventFlag					:= stStationEvents[4].aEvents[1].bEventTimer.Q;
stStationEvents[4].aEvents[1].bEventText					:= 'Process Door Retract timeout';
stStationEvents[4].aEvents[1].sSolution						:= 'Check cylinder, neumatic connections and sensors';





//CYCLE STOP REQUEST

(*stStationEvents[4].aEvents[2].bCycleStopRequest			:= TRUE;
stStationEvents[4].aEvents[2].bEventFlag					:= bEventsFlag[2];
stStationEvents[4].aEvents[2].bEventText					:= 'ST1 EVENT 7';*)
END_ACTION

END_PROGRAM

// ---- POUs/A_MASTER/A_2_PRG_MachineCtrl.TcPOU
PROGRAM A_2_PRG_MachineCtrl
VAR
/////////////////////////////////////////////////////////////////////////////////////TIMERS & TRIGGERS/////////////////////////////////////////////////////////////////////////////////////

	tonSys_Init					: Tc2_Standard.TON:=(PT:=T#1S);
	tonSys_InitTimeout			: Tc2_Standard.TON:=(PT:=T#15S);					
	tonFirstAutoCycle			: Tc2_Standard.TON:=(PT:=T#500MS);
	tonStopped					: TON := (PT := T#500MS);
	
/////////////////////////////////////////////////////////////////////////////////////PROCESS CYCLE/////////////////////////////////////////////////////////////////////////////////////	
	
	eCycleState					: E_General_ProcessCycle;
	tonCMD_Done					: TON;
	tonResetAllCMD				: TON;
	tonExecute					: TON;
	tonCylinderDwell			: TON; //Renan added - Buglist n13 - 08Jul26
	tonSave_Data				: TON;
	tonWriteToCsv				: TON;
	rFirstAutoCycle				: R_TRIG;
	
	bStartProcessCondition		: BOOL;
	i							: INT;
	j							: INT;
	
	bVisionProcessDoneFlag		: BOOL;
	tonGettingResults			: TON;
	tonWaitExtendCylidner		: TON;
	tonTakePicture				: TON;
	ctuRejectPart				: CTU;
	rRejectSensor				: R_TRIG;

/////////////////////////////////////////////////////////////////////////////////////SAFETY/////////////////////////////////////////////////////////////////////////////////////		
	



/////////////////////////////////////////////////////////////////////////////////////I/O/////////////////////////////////////////////////////////////////////////////////////	

	bPartPresentNest1			: BOOL;
	bPartPresentNest2			: BOOL;
	bPartPresentNest3			: BOOL;
	bPartPresentNest4			: BOOL;
	
	bTwoHandsSignal				: BOOL;
	tonTwoHandsSignal			: TON;
	
	bEndAutoCycleFlag			: BOOL;
	bProcessedPart				: ARRAY[0..1] OF BOOL;
	fProcessedPart				: ARRAY[0..1] OF F_TRIG;
	
	(* Renan Added - Buglist n6 - 08Jul26 *)
	bNest1StartOK				: BOOL;
	bNest2StartOK				: BOOL;
	bCycleHasFailure 			: BOOL;
	bCycleAllProcessedPass		: BOOL;
	(*\Renan Added - Buglist n6 - 08Jul26 *)
	
	bPuckLockerReadyToStart		: BOOL; (* Renan Added - Puck Locker Bug - 08Jul26 *)
	nPucksToRelease 			: USINT;(* Renan Added - Puck Locker Bug - 08Jul26 *)
	bPuckLockerEnable       	: BOOL; (* Renan added - Puck Locker Bug - 10Jul26*)
	
END_VAR

/////////////////////////////////////////////////////////////////////////////////////GENERAL/////////////////////////////////////////////////////////////////////////////////////
a_ACT_MachineStatus();
b_ACT_ProcessCycle();
d_ACT_IO();
e_ACT_SafetyProcess();

ACTION a_ACT_MachineStatus:
/////////////////////////////////////////////////////////////////////////////////////Utilities/////////////////////////////////////////////////////////////////////////////////////
tonSys_Init(IN:=stMachineStatus.bInitialising);
tonSafety( IN := stMachineStatus.eMachineState = E_MachineState.SAFETY, PT := T#10S);
tonStopped(IN := stMachineStatus.eMachineState = E_MachineState.STOPPED);
	
	IF stMachineStatus.eMachineState <> E_MachineState.SYSTEM_AUTO_CYCLE AND 
		stMachineStatus.eMachineState <> E_MachineState.SYSTEM_INITIALISING THEN
		
		sMachineMessage									:= '';			
		
	END_IF
	
	IF stMachineStatus.eMachineState <> E_MachineState.SYSTEM_INITIALISING THEN
		
		tonSys_InitTimeout.IN							:= FALSE;			
		
	END_IF
	
	IF (stMachineStatus.eMachineState = E_MachineState.STOPPED)  OR 
		(stMachineStatus.eMachineState = E_MachineState.STOPPING) THEN
		
		stTwinSAFE.iMachineStopped						:= TRUE;
		stTwinSAFE.iRunSafety							:= FALSE;
	
	ELSIF (stMachineStatus.eMachineState = E_MachineState.SAFETY) OR (stMachineStatus.eMachineState = E_MachineState.SYSTEM_INITIALISING) OR 
		(stMachineStatus.eMachineState = E_MachineState.SYSTEM_READY_TO_START) OR (stMachineStatus.eMachineState = E_MachineState.SYSTEM_AUTO_CYCLE) 
		OR (stMachineStatus.eMachineState = E_MachineState.MANUAL_MODE)THEN

		stTwinSAFE.iRunSafety							:= TRUE;
		stTwinSAFE.iMachineStopped						:= FALSE;
	
	ELSE stTwinSAFE.iMachineStopped						:= FALSE;
		stTwinSAFE.iRunSafety							:= FALSE;
		
	END_IF
	
	IF stMachineStatus.eMachineState = E_MachineState.SAFETY THEN
		
		stTwinSAFE.iInitSafety							:= TRUE;
		
	ELSE stTwinSAFE.iInitSafety							:= FALSE;
		
	END_IF

/////////////////////////////////////////////////////////////////////////////////////CONDITIONS/////////////////////////////////////////////////////////////////////////////////////
				IF NOT stMasterCtrl.bNoFault THEN
					stMachineStatus.eMachineState 		:= E_MachineState.FAULT;
				END_IF
				
				IF stMachineStatus.eMachineState		= E_MachineState.STOPPING OR
				stMachineStatus.eMachineState			= E_MachineState.FAULT THEN
					
					stCamera.CMD.bAbort					:= TRUE;	
					stLeakTesters.CMD.bAbort			:= TRUE;	
					stHeightTests.CMD.bAbort			:= TRUE;
					stProcessCylinder.CMD.bAbort		:= TRUE;
					stProcessDoor.CMD.bAbort			:= TRUE;
				
					stCamera.CMD.bEnable				:= FALSE;	
					stLeakTesters.CMD.bEnable			:= FALSE;	
					stHeightTests.CMD.bEnable			:= FALSE;
					stProcessCylinder.CMD.bEnable		:= FALSE;
					stProcessDoor.CMD.bEnable			:= FALSE;
					
				END_IF
				
				IF 	stButtonsLamps.bResetButtonFallingEdge THEN
					stCamera.CMD.bReset					:= TRUE;	
					stLeakTesters.CMD.bReset			:= TRUE;	
					stHeightTests.CMD.bReset			:= TRUE;
					stProcessCylinder.CMD.bReset		:= TRUE;
					stProcessDoor.CMD.bReset			:= TRUE;
				ELSE 
					stCamera.CMD.bReset					:= FALSE;	
					stLeakTesters.CMD.bReset			:= FALSE;	
					stHeightTests.CMD.bReset			:= FALSE;
					stProcessCylinder.CMD.bReset		:= FALSE;
					stProcessDoor.CMD.bReset			:= FALSE;
				END_IF

				IF 	NOT (stMachineStatus.eMachineState = E_MachineState.MANUAL_MODE) THEN
					
					stCamera.CMD.bManualMode				:=FALSE;
					stLeakTesters.CMD.bManualMode			:=FALSE;
					stHeightTests.CMD.bManualMode			:=FALSE;
					stProcessCylinder.CMD.bManualMode		:=FALSE;
					stProcessDoor.CMD.bManualMode			:=FALSE;
					
				END_IF
				
				IF stMachineStatus.eMachineState = E_MachineState.SYSTEM_POWER_UP THEN
					
					bReadAMSNetID							:= TRUE;
				
				ELSE 
					
					bReadAMSNetID							:= FALSE;
					
				END_IF;
				
				IF stMachineStatus.eMachineState		= E_MachineState.FAULT THEN
					
					bOpenDoorCycleFault						:= TRUE;
					
					
				ELSE bOpenDoorCycleFault					:= FALSE;
					
				END_IF
				
/////////////////////////////////////////////////////////////////////////////////////MACHINE CONTROL/////////////////////////////////////////////////////////////////////////////////////

CASE stMachineStatus.eMachineState OF

E_MachineState.SYSTEM_POWER_UP: 		

				fbGetLocalAMSNetID.bExecute				:= TRUE;
				bLightsOnOff							:= TRUE;
				IF tonSystemPowerUP.Q THEN
						stMachineStatus.eMachineState 	:= E_MachineState.STOPPED;
				END_IF
	
E_MachineState.STOPPED:		

				stTwinSAFE.iRunSafety					:= FALSE;				
				IF stMasterCtrl.bNoFault   AND NOT stMasterCtrl.bCycleStopRequest AND ftrigButton[3].Q AND tonStopped.Q THEN
						stMachineStatus.eMachineState 	:= E_MachineState.SAFETY;
				ELSIF NOT stMasterCtrl.bNoFault    THEN	
					stMachineStatus.eMachineState 		:= E_MachineState.FAULT;		
				END_IF

E_MachineState.SAFETY:

				GVL_IO.dw_T09_EL2809.qOpenProcessDoor   := TRUE; // Thays added - Buglist n1 - 08Jul26
				stTwinSAFE.iRunSafety					:= TRUE; 
				
				IF stTwinSAFE.qSafetyOk THEN
					
					stMachineStatus.eMachineState		:= E_MachineState.SYSTEM_INITIALISING;
					
				ELSIF stButtonsLamps.bStopButtonFallingEdge OR  
				stMasterCtrl.bCycleStopRequest OR tonSys_InitTimeout.Q  THEN
				
					stMachineStatus.eMachineState 		:= E_MachineState.STOPPING;	
					
				ELSIF NOT stMasterCtrl.bNoFault THEN		
					
					stMachineStatus.eMachineState 		:= E_MachineState.FAULT;
	
				END_IF
								

E_MachineState.SYSTEM_INITIALISING:		
					
					
				stCamera.CMD.bAbort						:= FALSE;	
				stLeakTesters.CMD.bAbort				:= FALSE;	
				stHeightTests.CMD.bAbort				:= FALSE;
				stProcessCylinder.CMD.bAbort			:= FALSE;
				stProcessDoor.CMD.bAbort				:= FALSE;
	

				IF tonSys_Init.Q THEN
					
					
					IF NOT stTwinSAFE.qProcessCylinderRetracted AND NOT bProcessDoorClosed THEN
						
						sMachineMessage					:= 'trigger both safety buttons to reset machine';
						
						IF bTwoHandsSignal THEN
							
							tonSys_InitTimeout.IN			:= TRUE;
							stCamera.CMD.bEnable			:= TRUE;	
							stLeakTesters.CMD.bEnable		:= TRUE;	
							stHeightTests.CMD.bEnable		:= TRUE;
							stProcessCylinder.CMD.bEnable	:= TRUE;
							stProcessDoor.CMD.bEnable		:= TRUE; 
							sMachineMessage					:= '';
							
						END_IF
					ELSE
						
						tonSys_InitTimeout.IN			:= TRUE;
						stCamera.CMD.bEnable			:= TRUE;	
						stLeakTesters.CMD.bEnable		:= TRUE;	
						stHeightTests.CMD.bEnable		:= TRUE;
						stProcessCylinder.CMD.bEnable	:= TRUE;
						stProcessDoor.CMD.bEnable		:= TRUE; 
						
					END_IF
											
				END_IF
				
				IF stMasterCtrl.bAllStationsReady  THEN 
					stMachineStatus.eMachineState		:= E_MachineState.SYSTEM_READY_TO_START;
				ELSIF stButtonsLamps.bStopButtonFallingEdge OR  
				stMasterCtrl.bCycleStopRequest OR tonSys_InitTimeout.Q  THEN
					stMachineStatus.eMachineState 		:= E_MachineState.STOPPING;	
				ELSIF NOT stMasterCtrl.bNoFault THEN		
					stMachineStatus.eMachineState 		:= E_MachineState.FAULT;
				END_IF;
			
					
E_MachineState.SYSTEM_READY_TO_START:			

				IF 	 stButtonsLamps.bStartButtonFallingEdge AND stMasterCtrl.bAllStationsReady  THEN
					stMachineStatus.eMachineState 		:= E_MachineState.SYSTEM_AUTO_CYCLE;
				ELSIF NOT stMasterCtrl.bAllStationsReady OR stMasterCtrl.bCycleStopRequest THEN
					stMachineStatus.eMachineState 		:= E_MachineState.STOPPING;		
				ELSIF NOT stMasterCtrl.bNoFault THEN	
					stMachineStatus.eMachineState 		:= E_MachineState.FAULT;
				ELSIF GVL_Master.stMasterCTRL.bManualModeRequest AND stMasterCtrl.bNoFault THEN
					stMachineStatus.eMachineState 		:= E_MachineState.MANUAL_MODE;
				END_IF

				

E_MachineState.SYSTEM_AUTO_CYCLE:		

				
				IF  stMasterCtrl.bCycleStopRequest AND (eCycleState = E_General_ProcessCycle.IDLE) THEN
	
					stMachineStatus.eMachineState 		:= E_MachineState.STOPPING;
				
				ELSIF stMasterCtrl.bCycleStopRequest AND NOT (eCycleState = E_General_ProcessCycle.IDLE) THEN					
				
					sMachineMessage						:= 'Ending  Cycle';
				
				ELSIF NOT stMasterCtrl.bNoFault THEN	
					stMachineStatus.eMachineState 		:= E_MachineState.FAULT;
				END_IF
				

E_MachineState.STOPPING:	

				
				IF stMasterCtrl.bAllStationsStopped THEN
					stMachineStatus.eMachineState 		:= E_MachineState.STOPPED;
				ELSIF NOT stMasterCtrl.bNoFault THEN	
					stMachineStatus.eMachineState 		:= E_MachineState.FAULT;					
				END_IF
			
				stTwinSAFE.iRunSafety					:= FALSE;	

E_MachineState.FAULT:	

				GVL_IO.dw_T09_EL2809.qOpenProcessDoor   :=TRUE; // Thays added - Buglist n1 - 08Jul26
 
				IF stMasterCtrl.bNoFault 	THEN
					stMachineStatus.eMachineState		:= E_MachineState.STOPPED;		
				END_IF
				
				stTwinSAFE.iRunSafety					:= FALSE;	

E_MachineState.MANUAL_MODE:

				IF stButtonsLamps.bStopButtonFallingEdge OR NOT GVL_Master.stMasterCTRL.bManualModeRequest THEN
					stMachineStatus.eMachineState 		:= E_MachineState.STOPPING;
				ELSIF  NOT stMasterCtrl.bNoFault THEN	
					stMachineStatus.eMachineState 		:= E_MachineState.FAULT;								
				ELSE 
					
					stCamera.CMD.bManualMode				:=TRUE;
					stLeakTesters.CMD.bManualMode			:=TRUE;
					stHeightTests.CMD.bManualMode			:=TRUE;
					stProcessCylinder.CMD.bManualMode		:=TRUE;
					stProcessDoor.CMD.bManualMode			:=TRUE;

				END_IF
				
					
ELSE
stMachineStatus.eMachineState:=E_MachineState.SYSTEM_POWER_UP;		
END_CASE									


